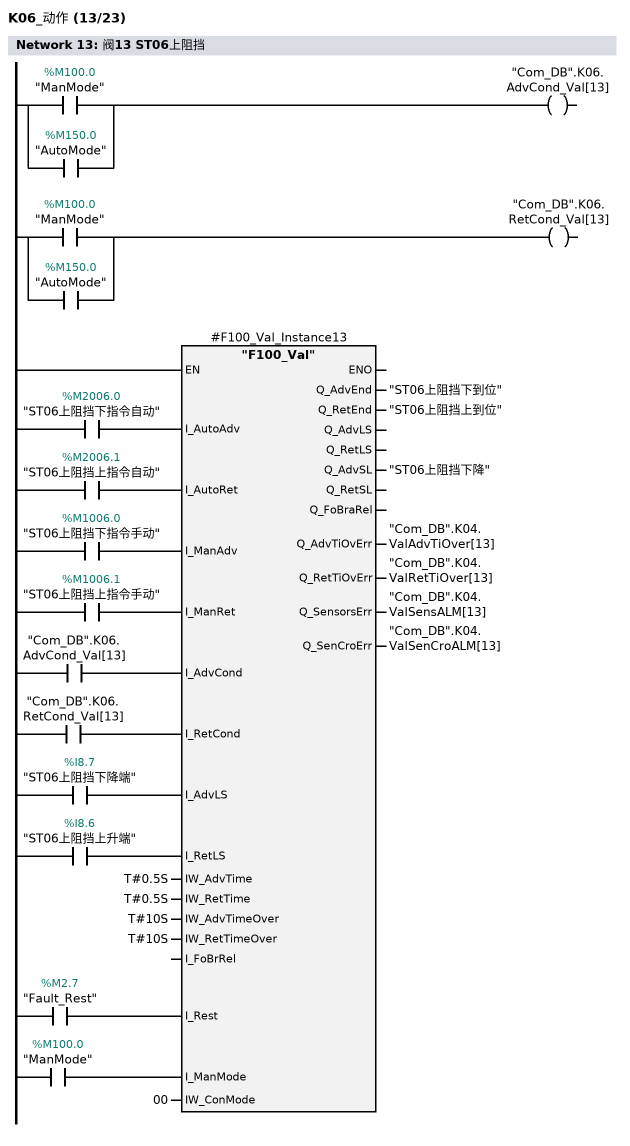
   RUNG wire#powerrail
      Contact( "ManMode" )
      wire#w1
      Coil( "Com_DB".K06.AdvCond_Val[13] )
   END_RUNG
   RUNG wire#powerrail
      Contact( "AutoMode" )
   END_RUNG wire#w1
   RUNG wire#powerrail
      Contact( "ManMode" )
      wire#w2
      Coil( "Com_DB".K06.RetCond_Val[13] )
   END_RUNG
   RUNG wire#powerrail
      Contact( "AutoMode" )
   END_RUNG wire#w2
   RUNG wire#powerrail
      #F100_Val_Instance13(I_AutoAdv := wire#w3, I_AutoRet := wire#w4, I_ManAdv := wire#w5, I_ManRet := wire#w6, I_AdvCond := wire#w7, I_RetCond := wire#w8, I_AdvLS := wire#w9, I_RetLS := wire#w10, I_Rest := wire#w11, I_ManMode := wire#w12, IW_AdvTime := T#0.5S, IW_RetTime := T#0.5S, IW_AdvTimeOver := T#10S, IW_RetTimeOver := T#10S, I_FoBrRel :=, IW_ConMode := 00, Q_AdvEnd => "ST06上阻挡下到位", Q_RetEnd => "ST06上阻挡上到位", Q_AdvLS =>, Q_RetLS =>, Q_AdvSL => "ST06上阻挡下降", Q_RetSL =>, Q_FoBraRel =>, Q_AdvTiOvErr => "Com_DB".K04.ValAdvTiOver[13], Q_RetTiOvErr => "Com_DB".K04.ValRetTiOver[13], Q_SensorsErr => "Com_DB".K04.ValSensALM[13], Q_SenCroErr => "Com_DB".K04.ValSenCroALM[13])
   END_RUNG
   RUNG wire#powerrail
      Contact( "ST06上阻挡下指令自动" )
   END_RUNG wire#w3
   RUNG wire#powerrail
      Contact( "ST06上阻挡上指令自动" )
   END_RUNG wire#w4
   RUNG wire#powerrail
      Contact( "ST06上阻挡下指令手动" )
   END_RUNG wire#w5
   RUNG wire#powerrail
      Contact( "ST06上阻挡上指令手动" )
   END_RUNG wire#w6
   RUNG wire#powerrail
      Contact( "Com_DB".K06.AdvCond_Val[13] )
   END_RUNG wire#w7
   RUNG wire#powerrail
      Contact( "Com_DB".K06.RetCond_Val[13] )
   END_RUNG wire#w8
   RUNG wire#powerrail
      Contact( "ST06上阻挡下降端" )
   END_RUNG wire#w9
   RUNG wire#powerrail
      Contact( "ST06上阻挡上升端" )
   END_RUNG wire#w10
   RUNG wire#powerrail
      Contact( "Fault_Rest" )
   END_RUNG wire#w11
   RUNG wire#powerrail
      Contact( "ManMode" )
   END_RUNG wire#w12
   // the same network as SCL:
   "Com_DB".K06.AdvCond_Val[13] := "ManMode" OR "AutoMode";
   "Com_DB".K06.RetCond_Val[13] := "ManMode" OR "AutoMode";
   #F100_Val_Instance13(I_AutoAdv := "ST06上阻挡下指令自动",   // "F100_Val"
                        I_AutoRet := "ST06上阻挡上指令自动",
                        I_ManAdv := "ST06上阻挡下指令手动",
                        I_ManRet := "ST06上阻挡上指令手动",
                        I_AdvCond := "Com_DB".K06.AdvCond_Val[13],
                        I_RetCond := "Com_DB".K06.RetCond_Val[13],
                        I_AdvLS := "ST06上阻挡下降端",
                        I_RetLS := "ST06上阻挡上升端",
                        IW_AdvTime := T#0.5S,
                        IW_RetTime := T#0.5S,
                        IW_AdvTimeOver := T#10S,
                        IW_RetTimeOver := T#10S,
                        I_Rest := "Fault_Rest",
                        I_ManMode := "ManMode",
                        IW_ConMode := 00,
                        Q_AdvEnd => "ST06上阻挡下到位",
                        Q_RetEnd => "ST06上阻挡上到位",
                        Q_AdvSL => "ST06上阻挡下降",
                        Q_AdvTiOvErr => "Com_DB".K04.ValAdvTiOver[13],
                        Q_RetTiOvErr => "Com_DB".K04.ValRetTiOver[13],
                        Q_SensorsErr => "Com_DB".K04.ValSensALM[13],
                        Q_SenCroErr => "Com_DB".K04.ValSenCroALM[13]);
END_REGION

REGION Network 14: 阀14 ST07上阻挡
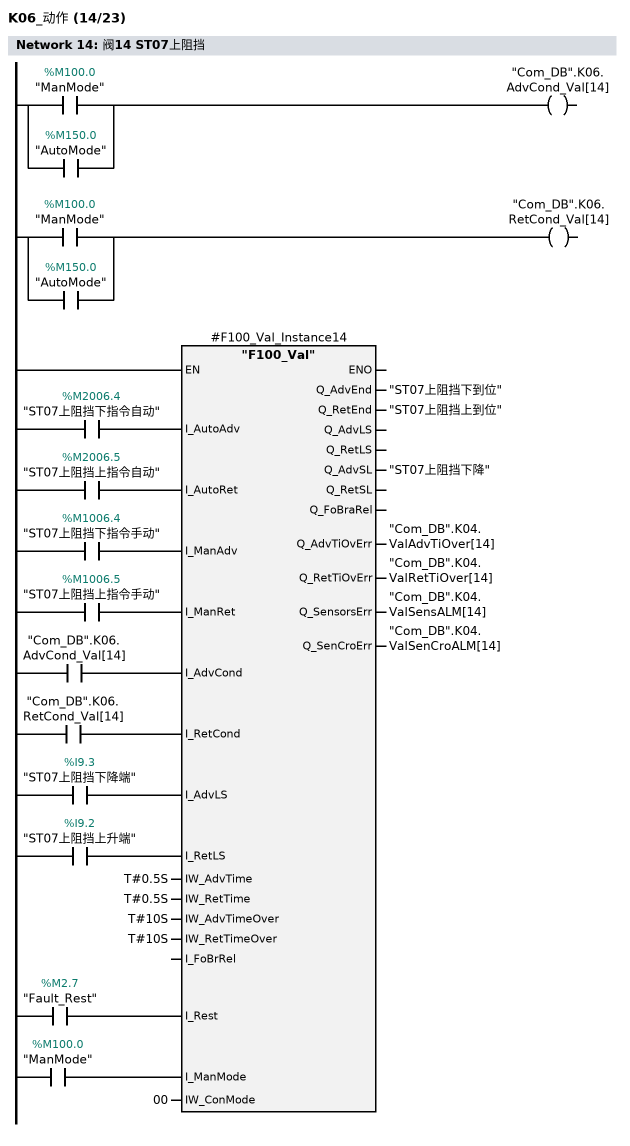
   RUNG wire#powerrail
      Contact( "ManMode" )
      wire#w1
      Coil( "Com_DB".K06.AdvCond_Val[14] )
   END_RUNG
   RUNG wire#powerrail
      Contact( "AutoMode" )
   END_RUNG wire#w1
   RUNG wire#powerrail
      Contact( "ManMode" )
      wire#w2
      Coil( "Com_DB".K06.RetCond_Val[14] )
   END_RUNG
   RUNG wire#powerrail
      Contact( "AutoMode" )
   END_RUNG wire#w2
   RUNG wire#powerrail
      #F100_Val_Instance14(I_AutoAdv := wire#w3, I_AutoRet := wire#w4, I_ManAdv := wire#w5, I_ManRet := wire#w6, I_AdvCond := wire#w7, I_RetCond := wire#w8, I_AdvLS := wire#w9, I_RetLS := wire#w10, I_Rest := wire#w11, I_ManMode := wire#w12, IW_AdvTime := T#0.5S, IW_RetTime := T#0.5S, IW_AdvTimeOver := T#10S, IW_RetTimeOver := T#10S, I_FoBrRel :=, IW_ConMode := 00, Q_AdvEnd => "ST07上阻挡下到位", Q_RetEnd => "ST07上阻挡上到位", Q_AdvLS =>, Q_RetLS =>, Q_AdvSL => "ST07上阻挡下降", Q_RetSL =>, Q_FoBraRel =>, Q_AdvTiOvErr => "Com_DB".K04.ValAdvTiOver[14], Q_RetTiOvErr => "Com_DB".K04.ValRetTiOver[14], Q_SensorsErr => "Com_DB".K04.ValSensALM[14], Q_SenCroErr => "Com_DB".K04.ValSenCroALM[14])
   END_RUNG
   RUNG wire#powerrail
      Contact( "ST07上阻挡下指令自动" )
   END_RUNG wire#w3
   RUNG wire#powerrail
      Contact( "ST07上阻挡上指令自动" )
   END_RUNG wire#w4
   RUNG wire#powerrail
      Contact( "ST07上阻挡下指令手动" )
   END_RUNG wire#w5
   RUNG wire#powerrail
      Contact( "ST07上阻挡上指令手动" )
   END_RUNG wire#w6
   RUNG wire#powerrail
      Contact( "Com_DB".K06.AdvCond_Val[14] )
   END_RUNG wire#w7
   RUNG wire#powerrail
      Contact( "Com_DB".K06.RetCond_Val[14] )
   END_RUNG wire#w8
   RUNG wire#powerrail
      Contact( "ST07上阻挡下降端" )
   END_RUNG wire#w9
   RUNG wire#powerrail
      Contact( "ST07上阻挡上升端" )
   END_RUNG wire#w10
   RUNG wire#powerrail
      Contact( "Fault_Rest" )
   END_RUNG wire#w11
   RUNG wire#powerrail
      Contact( "ManMode" )
   END_RUNG wire#w12
   // the same network as SCL:
   "Com_DB".K06.AdvCond_Val[14] := "ManMode" OR "AutoMode";
   "Com_DB".K06.RetCond_Val[14] := "ManMode" OR "AutoMode";
   #F100_Val_Instance14(I_AutoAdv := "ST07上阻挡下指令自动",   // "F100_Val"
                        I_AutoRet := "ST07上阻挡上指令自动",
                        I_ManAdv := "ST07上阻挡下指令手动",
                        I_ManRet := "ST07上阻挡上指令手动",
                        I_AdvCond := "Com_DB".K06.AdvCond_Val[14],
                        I_RetCond := "Com_DB".K06.RetCond_Val[14],
                        I_AdvLS := "ST07上阻挡下降端",
                        I_RetLS := "ST07上阻挡上升端",
                        IW_AdvTime := T#0.5S,
                        IW_RetTime := T#0.5S,
                        IW_AdvTimeOver := T#10S,
                        IW_RetTimeOver := T#10S,
                        I_Rest := "Fault_Rest",
                        I_ManMode := "ManMode",
                        IW_ConMode := 00,
                        Q_AdvEnd => "ST07上阻挡下到位",
                        Q_RetEnd => "ST07上阻挡上到位",
                        Q_AdvSL => "ST07上阻挡下降",
                        Q_AdvTiOvErr => "Com_DB".K04.ValAdvTiOver[14],
                        Q_RetTiOvErr => "Com_DB".K04.ValRetTiOver[14],
                        Q_SensorsErr => "Com_DB".K04.ValSensALM[14],
                        Q_SenCroErr => "Com_DB".K04.ValSenCroALM[14]);
END_REGION

REGION Network 15: 阀15 ST08上阻挡
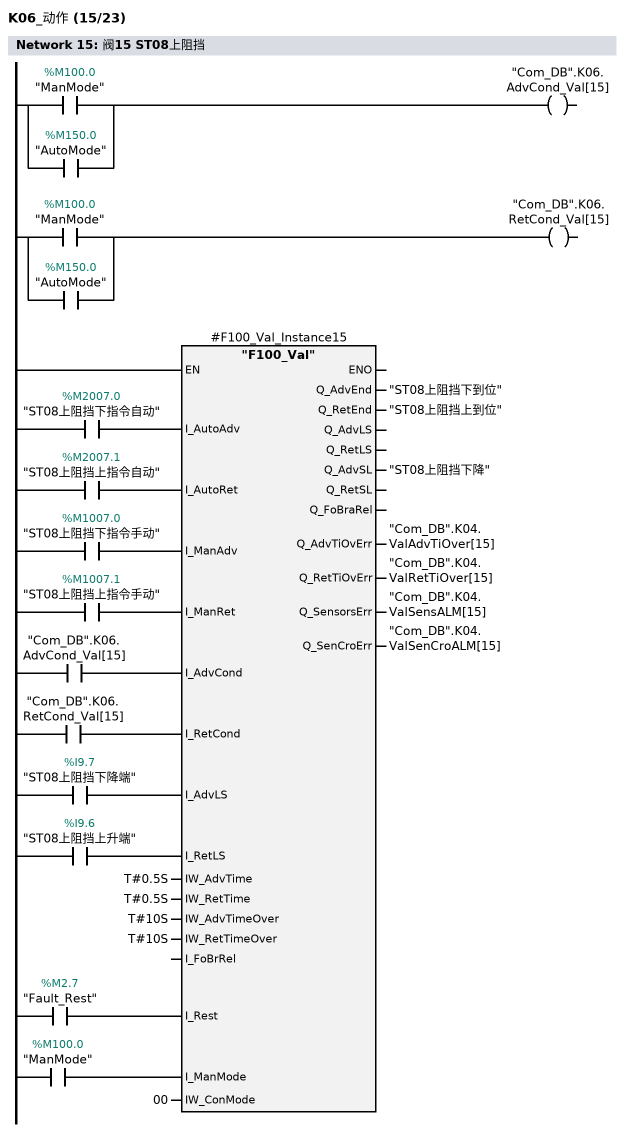
   RUNG wire#powerrail
      Contact( "ManMode" )
      wire#w1
      Coil( "Com_DB".K06.AdvCond_Val[15] )
   END_RUNG
   RUNG wire#powerrail
      Contact( "AutoMode" )
   END_RUNG wire#w1
   RUNG wire#powerrail
      Contact( "ManMode" )
      wire#w2
      Coil( "Com_DB".K06.RetCond_Val[15] )
   END_RUNG
   RUNG wire#powerrail
      Contact( "AutoMode" )
   END_RUNG wire#w2
   RUNG wire#powerrail
      #F100_Val_Instance15(I_AutoAdv := wire#w3, I_AutoRet := wire#w4, I_ManAdv := wire#w5, I_ManRet := wire#w6, I_AdvCond := wire#w7, I_RetCond := wire#w8, I_AdvLS := wire#w9, I_RetLS := wire#w10, I_Rest := wire#w11, I_ManMode := wire#w12, IW_AdvTime := T#0.5S, IW_RetTime := T#0.5S, IW_AdvTimeOver := T#10S, IW_RetTimeOver := T#10S, I_FoBrRel :=, IW_ConMode := 00, Q_AdvEnd => "ST08上阻挡下到位", Q_RetEnd => "ST08上阻挡上到位", Q_AdvLS =>, Q_RetLS =>, Q_AdvSL => "ST08上阻挡下降", Q_RetSL =>, Q_FoBraRel =>, Q_AdvTiOvErr => "Com_DB".K04.ValAdvTiOver[15], Q_RetTiOvErr => "Com_DB".K04.ValRetTiOver[15], Q_SensorsErr => "Com_DB".K04.ValSensALM[15], Q_SenCroErr => "Com_DB".K04.ValSenCroALM[15])
   END_RUNG
   RUNG wire#powerrail
      Contact( "ST08上阻挡下指令自动" )
   END_RUNG wire#w3
   RUNG wire#powerrail
      Contact( "ST08上阻挡上指令自动" )
   END_RUNG wire#w4
   RUNG wire#powerrail
      Contact( "ST08上阻挡下指令手动" )
   END_RUNG wire#w5
   RUNG wire#powerrail
      Contact( "ST08上阻挡上指令手动" )
   END_RUNG wire#w6
   RUNG wire#powerrail
      Contact( "Com_DB".K06.AdvCond_Val[15] )
   END_RUNG wire#w7
   RUNG wire#powerrail
      Contact( "Com_DB".K06.RetCond_Val[15] )
   END_RUNG wire#w8
   RUNG wire#powerrail
      Contact( "ST08上阻挡下降端" )
   END_RUNG wire#w9
   RUNG wire#powerrail
      Contact( "ST08上阻挡上升端" )
   END_RUNG wire#w10
   RUNG wire#powerrail
      Contact( "Fault_Rest" )
   END_RUNG wire#w11
   RUNG wire#powerrail
      Contact( "ManMode" )
   END_RUNG wire#w12
   // the same network as SCL:
   "Com_DB".K06.AdvCond_Val[15] := "ManMode" OR "AutoMode";
   "Com_DB".K06.RetCond_Val[15] := "ManMode" OR "AutoMode";
   #F100_Val_Instance15(I_AutoAdv := "ST08上阻挡下指令自动",   // "F100_Val"
                        I_AutoRet := "ST08上阻挡上指令自动",
                        I_ManAdv := "ST08上阻挡下指令手动",
                        I_ManRet := "ST08上阻挡上指令手动",
                        I_AdvCond := "Com_DB".K06.AdvCond_Val[15],
                        I_RetCond := "Com_DB".K06.RetCond_Val[15],
                        I_AdvLS := "ST08上阻挡下降端",
                        I_RetLS := "ST08上阻挡上升端",
                        IW_AdvTime := T#0.5S,
                        IW_RetTime := T#0.5S,
                        IW_AdvTimeOver := T#10S,
                        IW_RetTimeOver := T#10S,
                        I_Rest := "Fault_Rest",
                        I_ManMode := "ManMode",
                        IW_ConMode := 00,
                        Q_AdvEnd => "ST08上阻挡下到位",
                        Q_RetEnd => "ST08上阻挡上到位",
                        Q_AdvSL => "ST08上阻挡下降",
                        Q_AdvTiOvErr => "Com_DB".K04.ValAdvTiOver[15],
                        Q_RetTiOvErr => "Com_DB".K04.ValRetTiOver[15],
                        Q_SensorsErr => "Com_DB".K04.ValSensALM[15],
                        Q_SenCroErr => "Com_DB".K04.ValSenCroALM[15]);
END_REGION

REGION Network 16: 阀16 ST09上阻挡
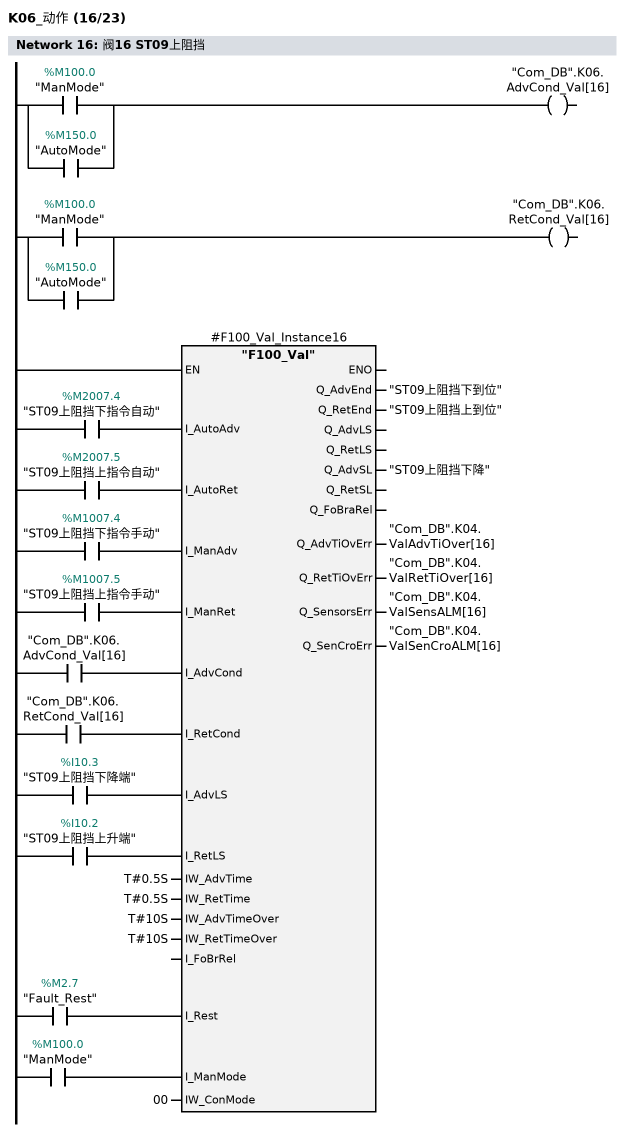
   RUNG wire#powerrail
      Contact( "ManMode" )
      wire#w1
      Coil( "Com_DB".K06.AdvCond_Val[16] )
   END_RUNG
   RUNG wire#powerrail
      Contact( "AutoMode" )
   END_RUNG wire#w1
   RUNG wire#powerrail
      Contact( "ManMode" )
      wire#w2
      Coil( "Com_DB".K06.RetCond_Val[16] )
   END_RUNG
   RUNG wire#powerrail
      Contact( "AutoMode" )
   END_RUNG wire#w2
   RUNG wire#powerrail
      #F100_Val_Instance16(I_AutoAdv := wire#w3, I_AutoRet := wire#w4, I_ManAdv := wire#w5, I_ManRet := wire#w6, I_AdvCond := wire#w7, I_RetCond := wire#w8, I_AdvLS := wire#w9, I_RetLS := wire#w10, I_Rest := wire#w11, I_ManMode := wire#w12, IW_AdvTime := T#0.5S, IW_RetTime := T#0.5S, IW_AdvTimeOver := T#10S, IW_RetTimeOver := T#10S, I_FoBrRel :=, IW_ConMode := 00, Q_AdvEnd => "ST09上阻挡下到位", Q_RetEnd => "ST09上阻挡上到位", Q_AdvLS =>, Q_RetLS =>, Q_AdvSL => "ST09上阻挡下降", Q_RetSL =>, Q_FoBraRel =>, Q_AdvTiOvErr => "Com_DB".K04.ValAdvTiOver[16], Q_RetTiOvErr => "Com_DB".K04.ValRetTiOver[16], Q_SensorsErr => "Com_DB".K04.ValSensALM[16], Q_SenCroErr => "Com_DB".K04.ValSenCroALM[16])
   END_RUNG
   RUNG wire#powerrail
      Contact( "ST09上阻挡下指令自动" )
   END_RUNG wire#w3
   RUNG wire#powerrail
      Contact( "ST09上阻挡上指令自动" )
   END_RUNG wire#w4
   RUNG wire#powerrail
      Contact( "ST09上阻挡下指令手动" )
   END_RUNG wire#w5
   RUNG wire#powerrail
      Contact( "ST09上阻挡上指令手动" )
   END_RUNG wire#w6
   RUNG wire#powerrail
      Contact( "Com_DB".K06.AdvCond_Val[16] )
   END_RUNG wire#w7
   RUNG wire#powerrail
      Contact( "Com_DB".K06.RetCond_Val[16] )
   END_RUNG wire#w8
   RUNG wire#powerrail
      Contact( "ST09上阻挡下降端" )
   END_RUNG wire#w9
   RUNG wire#powerrail
      Contact( "ST09上阻挡上升端" )
   END_RUNG wire#w10
   RUNG wire#powerrail
      Contact( "Fault_Rest" )
   END_RUNG wire#w11
   RUNG wire#powerrail
      Contact( "ManMode" )
   END_RUNG wire#w12
   // the same network as SCL:
   "Com_DB".K06.AdvCond_Val[16] := "ManMode" OR "AutoMode";
   "Com_DB".K06.RetCond_Val[16] := "ManMode" OR "AutoMode";
   #F100_Val_Instance16(I_AutoAdv := "ST09上阻挡下指令自动",   // "F100_Val"
                        I_AutoRet := "ST09上阻挡上指令自动",
                        I_ManAdv := "ST09上阻挡下指令手动",
                        I_ManRet := "ST09上阻挡上指令手动",
                        I_AdvCond := "Com_DB".K06.AdvCond_Val[16],
                        I_RetCond := "Com_DB".K06.RetCond_Val[16],
                        I_AdvLS := "ST09上阻挡下降端",
                        I_RetLS := "ST09上阻挡上升端",
                        IW_AdvTime := T#0.5S,
                        IW_RetTime := T#0.5S,
                        IW_AdvTimeOver := T#10S,
                        IW_RetTimeOver := T#10S,
                        I_Rest := "Fault_Rest",
                        I_ManMode := "ManMode",
                        IW_ConMode := 00,
                        Q_AdvEnd => "ST09上阻挡下到位",
                        Q_RetEnd => "ST09上阻挡上到位",
                        Q_AdvSL => "ST09上阻挡下降",
                        Q_AdvTiOvErr => "Com_DB".K04.ValAdvTiOver[16],
                        Q_RetTiOvErr => "Com_DB".K04.ValRetTiOver[16],
                        Q_SensorsErr => "Com_DB".K04.ValSensALM[16],
                        Q_SenCroErr => "Com_DB".K04.ValSenCroALM[16]);
END_REGION

REGION Network 17: 阀17 ST10上阻挡
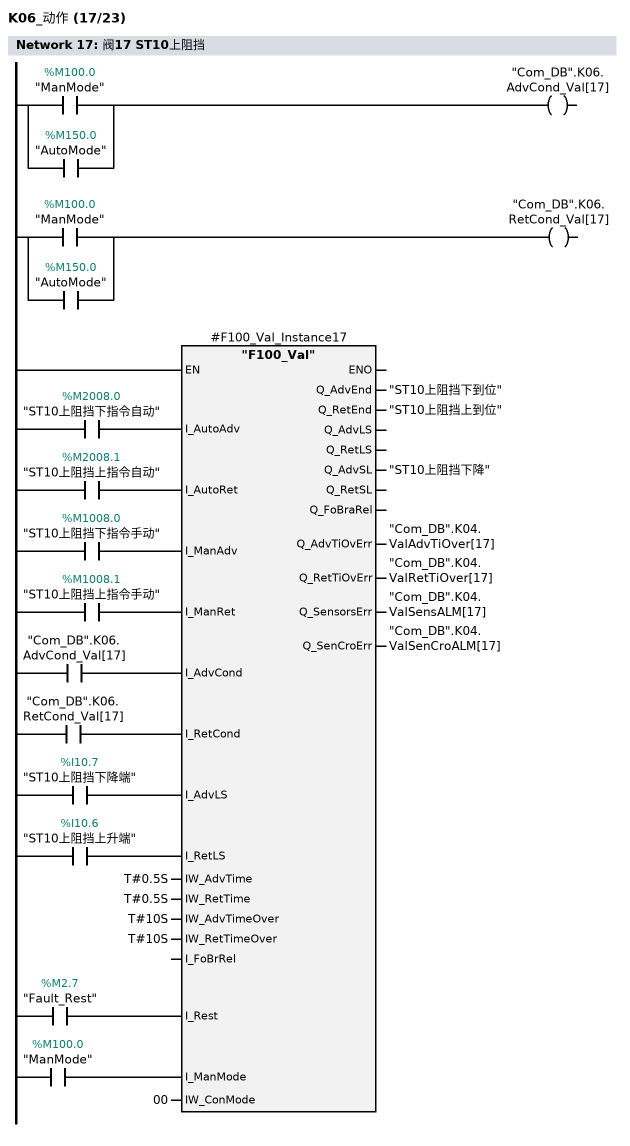
   RUNG wire#powerrail
      Contact( "ManMode" )
      wire#w1
      Coil( "Com_DB".K06.AdvCond_Val[17] )
   END_RUNG
   RUNG wire#powerrail
      Contact( "AutoMode" )
   END_RUNG wire#w1
   RUNG wire#powerrail
      Contact( "ManMode" )
      wire#w2
      Coil( "Com_DB".K06.RetCond_Val[17] )
   END_RUNG
   RUNG wire#powerrail
      Contact( "AutoMode" )
   END_RUNG wire#w2
   RUNG wire#powerrail
      #F100_Val_Instance17(I_AutoAdv := wire#w3, I_AutoRet := wire#w4, I_ManAdv := wire#w5, I_ManRet := wire#w6, I_AdvCond := wire#w7, I_RetCond := wire#w8, I_AdvLS := wire#w9, I_RetLS := wire#w10, I_Rest := wire#w11, I_ManMode := wire#w12, IW_AdvTime := T#0.5S, IW_RetTime := T#0.5S, IW_AdvTimeOver := T#10S, IW_RetTimeOver := T#10S, I_FoBrRel :=, IW_ConMode := 00, Q_AdvEnd => "ST10上阻挡下到位", Q_RetEnd => "ST10上阻挡上到位", Q_AdvLS =>, Q_RetLS =>, Q_AdvSL => "ST10上阻挡下降", Q_RetSL =>, Q_FoBraRel =>, Q_AdvTiOvErr => "Com_DB".K04.ValAdvTiOver[17], Q_RetTiOvErr => "Com_DB".K04.ValRetTiOver[17], Q_SensorsErr => "Com_DB".K04.ValSensALM[17], Q_SenCroErr => "Com_DB".K04.ValSenCroALM[17])
   END_RUNG
   RUNG wire#powerrail
      Contact( "ST10上阻挡下指令自动" )
   END_RUNG wire#w3
   RUNG wire#powerrail
      Contact( "ST10上阻挡上指令自动" )
   END_RUNG wire#w4
   RUNG wire#powerrail
      Contact( "ST10上阻挡下指令手动" )
   END_RUNG wire#w5
   RUNG wire#powerrail
      Contact( "ST10上阻挡上指令手动" )
   END_RUNG wire#w6
   RUNG wire#powerrail
      Contact( "Com_DB".K06.AdvCond_Val[17] )
   END_RUNG wire#w7
   RUNG wire#powerrail
      Contact( "Com_DB".K06.RetCond_Val[17] )
   END_RUNG wire#w8
   RUNG wire#powerrail
      Contact( "ST10上阻挡下降端" )
   END_RUNG wire#w9
   RUNG wire#powerrail
      Contact( "ST10上阻挡上升端" )
   END_RUNG wire#w10
   RUNG wire#powerrail
      Contact( "Fault_Rest" )
   END_RUNG wire#w11
   RUNG wire#powerrail
      Contact( "ManMode" )
   END_RUNG wire#w12
   // the same network as SCL:
   "Com_DB".K06.AdvCond_Val[17] := "ManMode" OR "AutoMode";
   "Com_DB".K06.RetCond_Val[17] := "ManMode" OR "AutoMode";
   #F100_Val_Instance17(I_AutoAdv := "ST10上阻挡下指令自动",   // "F100_Val"
                        I_AutoRet := "ST10上阻挡上指令自动",
                        I_ManAdv := "ST10上阻挡下指令手动",
                        I_ManRet := "ST10上阻挡上指令手动",
                        I_AdvCond := "Com_DB".K06.AdvCond_Val[17],
                        I_RetCond := "Com_DB".K06.RetCond_Val[17],
                        I_AdvLS := "ST10上阻挡下降端",
                        I_RetLS := "ST10上阻挡上升端",
                        IW_AdvTime := T#0.5S,
                        IW_RetTime := T#0.5S,
                        IW_AdvTimeOver := T#10S,
                        IW_RetTimeOver := T#10S,
                        I_Rest := "Fault_Rest",
                        I_ManMode := "ManMode",
                        IW_ConMode := 00,
                        Q_AdvEnd => "ST10上阻挡下到位",
                        Q_RetEnd => "ST10上阻挡上到位",
                        Q_AdvSL => "ST10上阻挡下降",
                        Q_AdvTiOvErr => "Com_DB".K04.ValAdvTiOver[17],
                        Q_RetTiOvErr => "Com_DB".K04.ValRetTiOver[17],
                        Q_SensorsErr => "Com_DB".K04.ValSensALM[17],
                        Q_SenCroErr => "Com_DB".K04.ValSenCroALM[17]);
END_REGION

REGION Network 18: 阀18 ST11上阻挡
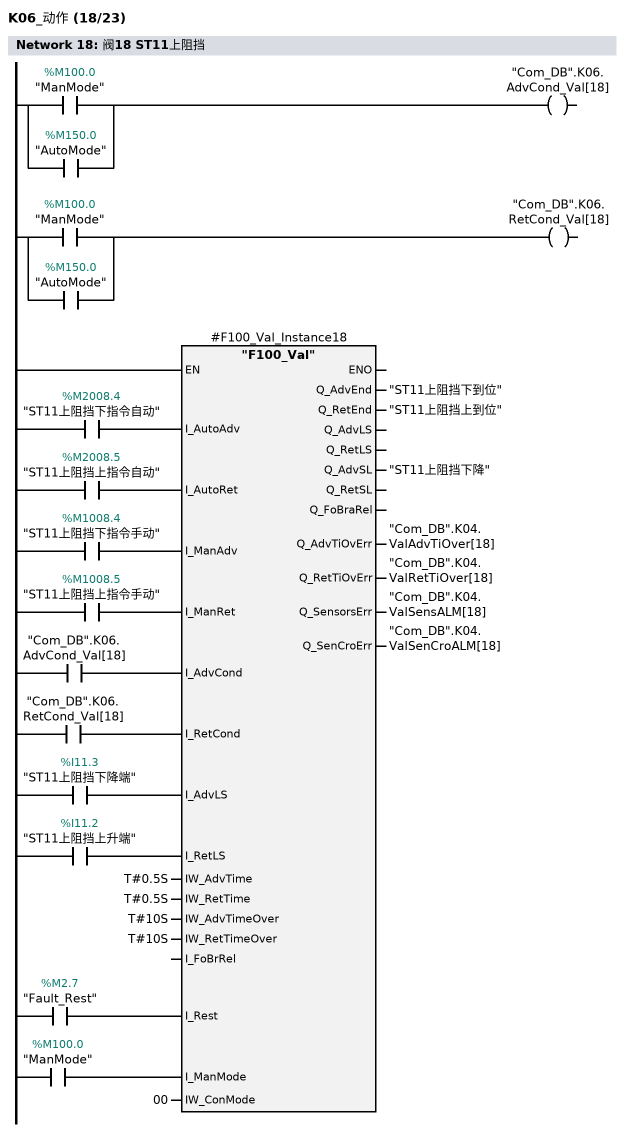
   RUNG wire#powerrail
      Contact( "ManMode" )
      wire#w1
      Coil( "Com_DB".K06.AdvCond_Val[18] )
   END_RUNG
   RUNG wire#powerrail
      Contact( "AutoMode" )
   END_RUNG wire#w1
   RUNG wire#powerrail
      Contact( "ManMode" )
      wire#w2
      Coil( "Com_DB".K06.RetCond_Val[18] )
   END_RUNG
   RUNG wire#powerrail
      Contact( "AutoMode" )
   END_RUNG wire#w2
   RUNG wire#powerrail
      #F100_Val_Instance18(I_AutoAdv := wire#w3, I_AutoRet := wire#w4, I_ManAdv := wire#w5, I_ManRet := wire#w6, I_AdvCond := wire#w7, I_RetCond := wire#w8, I_AdvLS := wire#w9, I_RetLS := wire#w10, I_Rest := wire#w11, I_ManMode := wire#w12, IW_AdvTime := T#0.5S, IW_RetTime := T#0.5S, IW_AdvTimeOver := T#10S, IW_RetTimeOver := T#10S, I_FoBrRel :=, IW_ConMode := 00, Q_AdvEnd => "ST11上阻挡下到位", Q_RetEnd => "ST11上阻挡上到位", Q_AdvLS =>, Q_RetLS =>, Q_AdvSL => "ST11上阻挡下降", Q_RetSL =>, Q_FoBraRel =>, Q_AdvTiOvErr => "Com_DB".K04.ValAdvTiOver[18], Q_RetTiOvErr => "Com_DB".K04.ValRetTiOver[18], Q_SensorsErr => "Com_DB".K04.ValSensALM[18], Q_SenCroErr => "Com_DB".K04.ValSenCroALM[18])
   END_RUNG
   RUNG wire#powerrail
      Contact( "ST11上阻挡下指令自动" )
   END_RUNG wire#w3
   RUNG wire#powerrail
      Contact( "ST11上阻挡上指令自动" )
   END_RUNG wire#w4
   RUNG wire#powerrail
      Contact( "ST11上阻挡下指令手动" )
   END_RUNG wire#w5
   RUNG wire#powerrail
      Contact( "ST11上阻挡上指令手动" )
   END_RUNG wire#w6
   RUNG wire#powerrail
      Contact( "Com_DB".K06.AdvCond_Val[18] )
   END_RUNG wire#w7
   RUNG wire#powerrail
      Contact( "Com_DB".K06.RetCond_Val[18] )
   END_RUNG wire#w8
   RUNG wire#powerrail
      Contact( "ST11上阻挡下降端" )
   END_RUNG wire#w9
   RUNG wire#powerrail
      Contact( "ST11上阻挡上升端" )
   END_RUNG wire#w10
   RUNG wire#powerrail
      Contact( "Fault_Rest" )
   END_RUNG wire#w11
   RUNG wire#powerrail
      Contact( "ManMode" )
   END_RUNG wire#w12
   // the same network as SCL:
   "Com_DB".K06.AdvCond_Val[18] := "ManMode" OR "AutoMode";
   "Com_DB".K06.RetCond_Val[18] := "ManMode" OR "AutoMode";
   #F100_Val_Instance18(I_AutoAdv := "ST11上阻挡下指令自动",   // "F100_Val"
                        I_AutoRet := "ST11上阻挡上指令自动",
                        I_ManAdv := "ST11上阻挡下指令手动",
                        I_ManRet := "ST11上阻挡上指令手动",
                        I_AdvCond := "Com_DB".K06.AdvCond_Val[18],
                        I_RetCond := "Com_DB".K06.RetCond_Val[18],
                        I_AdvLS := "ST11上阻挡下降端",
                        I_RetLS := "ST11上阻挡上升端",
                        IW_AdvTime := T#0.5S,
                        IW_RetTime := T#0.5S,
                        IW_AdvTimeOver := T#10S,
                        IW_RetTimeOver := T#10S,
                        I_Rest := "Fault_Rest",
                        I_ManMode := "ManMode",
                        IW_ConMode := 00,
                        Q_AdvEnd => "ST11上阻挡下到位",
                        Q_RetEnd => "ST11上阻挡上到位",
                        Q_AdvSL => "ST11上阻挡下降",
                        Q_AdvTiOvErr => "Com_DB".K04.ValAdvTiOver[18],
                        Q_RetTiOvErr => "Com_DB".K04.ValRetTiOver[18],
                        Q_SensorsErr => "Com_DB".K04.ValSensALM[18],
                        Q_SenCroErr => "Com_DB".K04.ValSenCroALM[18]);
END_REGION

REGION Network 19: 阀19 ST12上阻挡
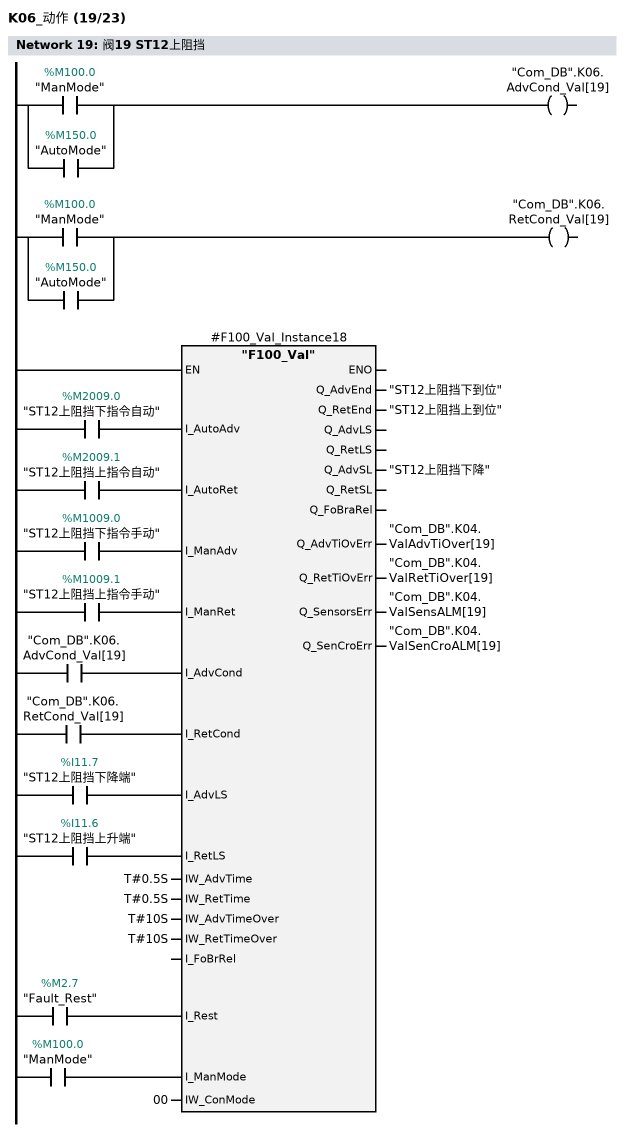
   RUNG wire#powerrail
      Contact( "ManMode" )
      wire#w1
      Coil( "Com_DB".K06.AdvCond_Val[19] )
   END_RUNG
   RUNG wire#powerrail
      Contact( "AutoMode" )
   END_RUNG wire#w1
   RUNG wire#powerrail
      Contact( "ManMode" )
      wire#w2
      Coil( "Com_DB".K06.RetCond_Val[19] )
   END_RUNG
   RUNG wire#powerrail
      Contact( "AutoMode" )
   END_RUNG wire#w2
   RUNG wire#powerrail
      #F100_Val_Instance18(I_AutoAdv := wire#w3, I_AutoRet := wire#w4, I_ManAdv := wire#w5, I_ManRet := wire#w6, I_AdvCond := wire#w7, I_RetCond := wire#w8, I_AdvLS := wire#w9, I_RetLS := wire#w10, I_Rest := wire#w11, I_ManMode := wire#w12, IW_AdvTime := T#0.5S, IW_RetTime := T#0.5S, IW_AdvTimeOver := T#10S, IW_RetTimeOver := T#10S, I_FoBrRel :=, IW_ConMode := 00, Q_AdvEnd => "ST12上阻挡下到位", Q_RetEnd => "ST12上阻挡上到位", Q_AdvLS =>, Q_RetLS =>, Q_AdvSL => "ST12上阻挡下降", Q_RetSL =>, Q_FoBraRel =>, Q_AdvTiOvErr => "Com_DB".K04.ValAdvTiOver[19], Q_RetTiOvErr => "Com_DB".K04.ValRetTiOver[19], Q_SensorsErr => "Com_DB".K04.ValSensALM[19], Q_SenCroErr => "Com_DB".K04.ValSenCroALM[19])
   END_RUNG
   RUNG wire#powerrail
      Contact( "ST12上阻挡下指令自动" )
   END_RUNG wire#w3
   RUNG wire#powerrail
      Contact( "ST12上阻挡上指令自动" )
   END_RUNG wire#w4
   RUNG wire#powerrail
      Contact( "ST12上阻挡下指令手动" )
   END_RUNG wire#w5
   RUNG wire#powerrail
      Contact( "ST12上阻挡上指令手动" )
   END_RUNG wire#w6
   RUNG wire#powerrail
      Contact( "Com_DB".K06.AdvCond_Val[19] )
   END_RUNG wire#w7
   RUNG wire#powerrail
      Contact( "Com_DB".K06.RetCond_Val[19] )
   END_RUNG wire#w8
   RUNG wire#powerrail
      Contact( "ST12上阻挡下降端" )
   END_RUNG wire#w9
   RUNG wire#powerrail
      Contact( "ST12上阻挡上升端" )
   END_RUNG wire#w10
   RUNG wire#powerrail
      Contact( "Fault_Rest" )
   END_RUNG wire#w11
   RUNG wire#powerrail
      Contact( "ManMode" )
   END_RUNG wire#w12
   // the same network as SCL:
   "Com_DB".K06.AdvCond_Val[19] := "ManMode" OR "AutoMode";
   "Com_DB".K06.RetCond_Val[19] := "ManMode" OR "AutoMode";
   #F100_Val_Instance18(I_AutoAdv := "ST12上阻挡下指令自动",   // "F100_Val"
                        I_AutoRet := "ST12上阻挡上指令自动",
                        I_ManAdv := "ST12上阻挡下指令手动",
                        I_ManRet := "ST12上阻挡上指令手动",
                        I_AdvCond := "Com_DB".K06.AdvCond_Val[19],
                        I_RetCond := "Com_DB".K06.RetCond_Val[19],
                        I_AdvLS := "ST12上阻挡下降端",
                        I_RetLS := "ST12上阻挡上升端",
                        IW_AdvTime := T#0.5S,
                        IW_RetTime := T#0.5S,
                        IW_AdvTimeOver := T#10S,
                        IW_RetTimeOver := T#10S,
                        I_Rest := "Fault_Rest",
                        I_ManMode := "ManMode",
                        IW_ConMode := 00,
                        Q_AdvEnd => "ST12上阻挡下到位",
                        Q_RetEnd => "ST12上阻挡上到位",
                        Q_AdvSL => "ST12上阻挡下降",
                        Q_AdvTiOvErr => "Com_DB".K04.ValAdvTiOver[19],
                        Q_RetTiOvErr => "Com_DB".K04.ValRetTiOver[19],
                        Q_SensorsErr => "Com_DB".K04.ValSensALM[19],
                        Q_SenCroErr => "Com_DB".K04.ValSenCroALM[19]);
END_REGION

REGION Network 20: 变频器1-入口搬送电机
   // 滚筒控制也可以使用变频器FB库，正转上层送托盘，反转下层接托盘
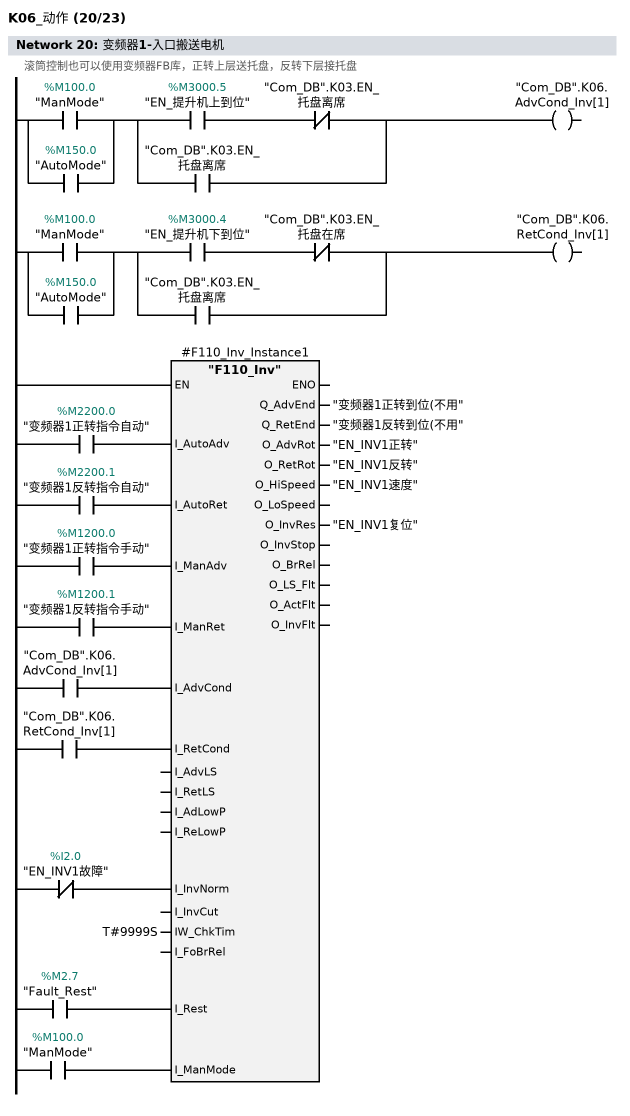
   RUNG wire#powerrail
      Contact( "ManMode" )
      wire#w1
      Contact( "EN_提升机上到位" )
      I_Contact( "Com_DB".K03.EN_托盘离席 )
      wire#w2
      Coil( "Com_DB".K06.AdvCond_Inv[1] )
   END_RUNG
   RUNG wire#powerrail
      Contact( "AutoMode" )
   END_RUNG wire#w1
   RUNG wire#w1
      Contact( "Com_DB".K03.EN_托盘离席 )
   END_RUNG wire#w2
   RUNG wire#powerrail
      Contact( "ManMode" )
      wire#w3
      Contact( "EN_提升机下到位" )
      I_Contact( "Com_DB".K03.EN_托盘在席 )
      wire#w4
      Coil( "Com_DB".K06.RetCond_Inv[1] )
   END_RUNG
   RUNG wire#powerrail
      Contact( "AutoMode" )
   END_RUNG wire#w3
   RUNG wire#w3
      Contact( "Com_DB".K03.EN_托盘离席 )
   END_RUNG wire#w4
   RUNG wire#powerrail
      #F110_Inv_Instance1(I_AutoAdv := wire#w5, I_AutoRet := wire#w6, I_ManAdv := wire#w7, I_ManRet := wire#w8, I_AdvCond := wire#w9, I_RetCond := wire#w10, I_InvNorm := wire#w11, I_Rest := wire#w12, I_ManMode := wire#w13, I_AdvLS :=, I_RetLS :=, I_AdLowP :=, I_ReLowP :=, I_InvCut :=, IW_ChkTim := T#9999S, I_FoBrRel :=, Q_AdvEnd => "变频器1正转到位(不用", Q_RetEnd => "变频器1反转到位(不用", O_AdvRot => "EN_INV1正转", O_RetRot => "EN_INV1反转", O_HiSpeed => "EN_INV1速度", O_LoSpeed =>, O_InvRes => "EN_INV1复位", O_InvStop =>, O_BrRel =>, O_LS_Flt =>, O_ActFlt =>, O_InvFlt =>)
   END_RUNG
   RUNG wire#powerrail
      Contact( "变频器1正转指令自动" )
   END_RUNG wire#w5
   RUNG wire#powerrail
      Contact( "变频器1反转指令自动" )
   END_RUNG wire#w6
   RUNG wire#powerrail
      Contact( "变频器1正转指令手动" )
   END_RUNG wire#w7
   RUNG wire#powerrail
      Contact( "变频器1反转指令手动" )
   END_RUNG wire#w8
   RUNG wire#powerrail
      Contact( "Com_DB".K06.AdvCond_Inv[1] )
   END_RUNG wire#w9
   RUNG wire#powerrail
      Contact( "Com_DB".K06.RetCond_Inv[1] )
   END_RUNG wire#w10
   RUNG wire#powerrail
      I_Contact( "EN_INV1故障" )
   END_RUNG wire#w11
   RUNG wire#powerrail
      Contact( "Fault_Rest" )
   END_RUNG wire#w12
   RUNG wire#powerrail
      Contact( "ManMode" )
   END_RUNG wire#w13
   // the same network as SCL:
   "Com_DB".K06.AdvCond_Inv[1] := ("ManMode" OR "AutoMode") AND (("EN_提升机上到位" AND NOT "Com_DB".K03.EN_托盘离席) OR "Com_DB".K03.EN_托盘离席);
   "Com_DB".K06.RetCond_Inv[1] := ("ManMode" OR "AutoMode") AND (("EN_提升机下到位" AND NOT "Com_DB".K03.EN_托盘在席) OR "Com_DB".K03.EN_托盘离席);
   #F110_Inv_Instance1(I_AutoAdv := "变频器1正转指令自动",   // "F110_Inv"
                       I_AutoRet := "变频器1反转指令自动",
                       I_ManAdv := "变频器1正转指令手动",
                       I_ManRet := "变频器1反转指令手动",
                       I_AdvCond := "Com_DB".K06.AdvCond_Inv[1],
                       I_RetCond := "Com_DB".K06.RetCond_Inv[1],
                       I_InvNorm := NOT "EN_INV1故障",
                       IW_ChkTim := T#9999S,
                       I_Rest := "Fault_Rest",
                       I_ManMode := "ManMode",
                       Q_AdvEnd => "变频器1正转到位(不用",
                       Q_RetEnd => "变频器1反转到位(不用",
                       O_AdvRot => "EN_INV1正转",
                       O_RetRot => "EN_INV1反转",
                       O_HiSpeed => "EN_INV1速度",
                       O_InvRes => "EN_INV1复位");
END_REGION

REGION Network 21: 变频器2 出口搬送电机
   // 正转上层J接托盘，反转下层送托盘
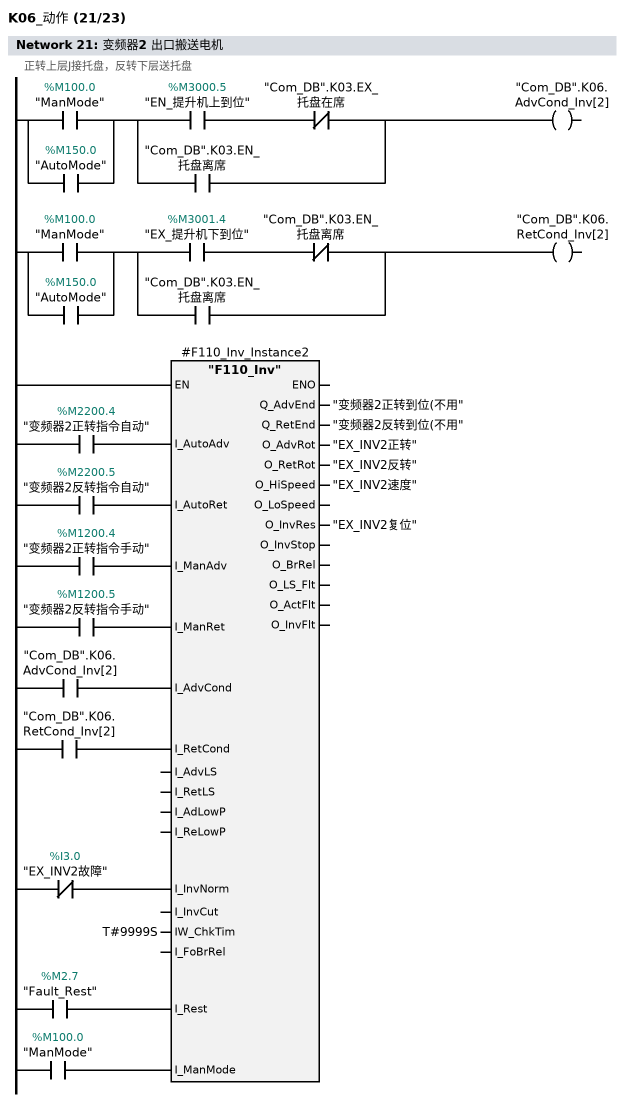
   RUNG wire#powerrail
      Contact( "ManMode" )
      wire#w1
      Contact( "EN_提升机上到位" )
      I_Contact( "Com_DB".K03.EX_托盘在席 )
      wire#w2
      Coil( "Com_DB".K06.AdvCond_Inv[2] )
   END_RUNG
   RUNG wire#powerrail
      Contact( "AutoMode" )
   END_RUNG wire#w1
   RUNG wire#w1
      Contact( "Com_DB".K03.EN_托盘离席 )
   END_RUNG wire#w2
   RUNG wire#powerrail
      Contact( "ManMode" )
      wire#w3
      Contact( "EX_提升机下到位" )
      I_Contact( "Com_DB".K03.EN_托盘离席 )
      wire#w4
      Coil( "Com_DB".K06.RetCond_Inv[2] )
   END_RUNG
   RUNG wire#powerrail
      Contact( "AutoMode" )
   END_RUNG wire#w3
   RUNG wire#w3
      Contact( "Com_DB".K03.EN_托盘离席 )
   END_RUNG wire#w4
   RUNG wire#powerrail
      #F110_Inv_Instance2(I_AutoAdv := wire#w5, I_AutoRet := wire#w6, I_ManAdv := wire#w7, I_ManRet := wire#w8, I_AdvCond := wire#w9, I_RetCond := wire#w10, I_InvNorm := wire#w11, I_Rest := wire#w12, I_ManMode := wire#w13, I_AdvLS :=, I_RetLS :=, I_AdLowP :=, I_ReLowP :=, I_InvCut :=, IW_ChkTim := T#9999S, I_FoBrRel :=, Q_AdvEnd => "变频器2正转到位(不用", Q_RetEnd => "变频器2反转到位(不用", O_AdvRot => "EX_INV2正转", O_RetRot => "EX_INV2反转", O_HiSpeed => "EX_INV2速度", O_LoSpeed =>, O_InvRes => "EX_INV2复位", O_InvStop =>, O_BrRel =>, O_LS_Flt =>, O_ActFlt =>, O_InvFlt =>)
   END_RUNG
   RUNG wire#powerrail
      Contact( "变频器2正转指令自动" )
   END_RUNG wire#w5
   RUNG wire#powerrail
      Contact( "变频器2反转指令自动" )
   END_RUNG wire#w6
   RUNG wire#powerrail
      Contact( "变频器2正转指令手动" )
   END_RUNG wire#w7
   RUNG wire#powerrail
      Contact( "变频器2反转指令手动" )
   END_RUNG wire#w8
   RUNG wire#powerrail
      Contact( "Com_DB".K06.AdvCond_Inv[2] )
   END_RUNG wire#w9
   RUNG wire#powerrail
      Contact( "Com_DB".K06.RetCond_Inv[2] )
   END_RUNG wire#w10
   RUNG wire#powerrail
      I_Contact( "EX_INV2故障" )
   END_RUNG wire#w11
   RUNG wire#powerrail
      Contact( "Fault_Rest" )
   END_RUNG wire#w12
   RUNG wire#powerrail
      Contact( "ManMode" )
   END_RUNG wire#w13
   // the same network as SCL:
   "Com_DB".K06.AdvCond_Inv[2] := ("ManMode" OR "AutoMode") AND (("EN_提升机上到位" AND NOT "Com_DB".K03.EX_托盘在席) OR "Com_DB".K03.EN_托盘离席);
   "Com_DB".K06.RetCond_Inv[2] := ("ManMode" OR "AutoMode") AND (("EX_提升机下到位" AND NOT "Com_DB".K03.EN_托盘离席) OR "Com_DB".K03.EN_托盘离席);
   #F110_Inv_Instance2(I_AutoAdv := "变频器2正转指令自动",   // "F110_Inv"
                       I_AutoRet := "变频器2反转指令自动",
                       I_ManAdv := "变频器2正转指令手动",
                       I_ManRet := "变频器2反转指令手动",
                       I_AdvCond := "Com_DB".K06.AdvCond_Inv[2],
                       I_RetCond := "Com_DB".K06.RetCond_Inv[2],
                       I_InvNorm := NOT "EX_INV2故障",
                       IW_ChkTim := T#9999S,
                       I_Rest := "Fault_Rest",
                       I_ManMode := "ManMode",
                       Q_AdvEnd => "变频器2正转到位(不用",
                       Q_RetEnd => "变频器2反转到位(不用",
                       O_AdvRot => "EX_INV2正转",
                       O_RetRot => "EX_INV2反转",
                       O_HiSpeed => "EX_INV2速度",
                       O_InvRes => "EX_INV2复位");
END_REGION

REGION Network 22: 变频器3/5 前段/后段上层搬送电机，因为上层变频器条件一致，功能一致。共用1个FB
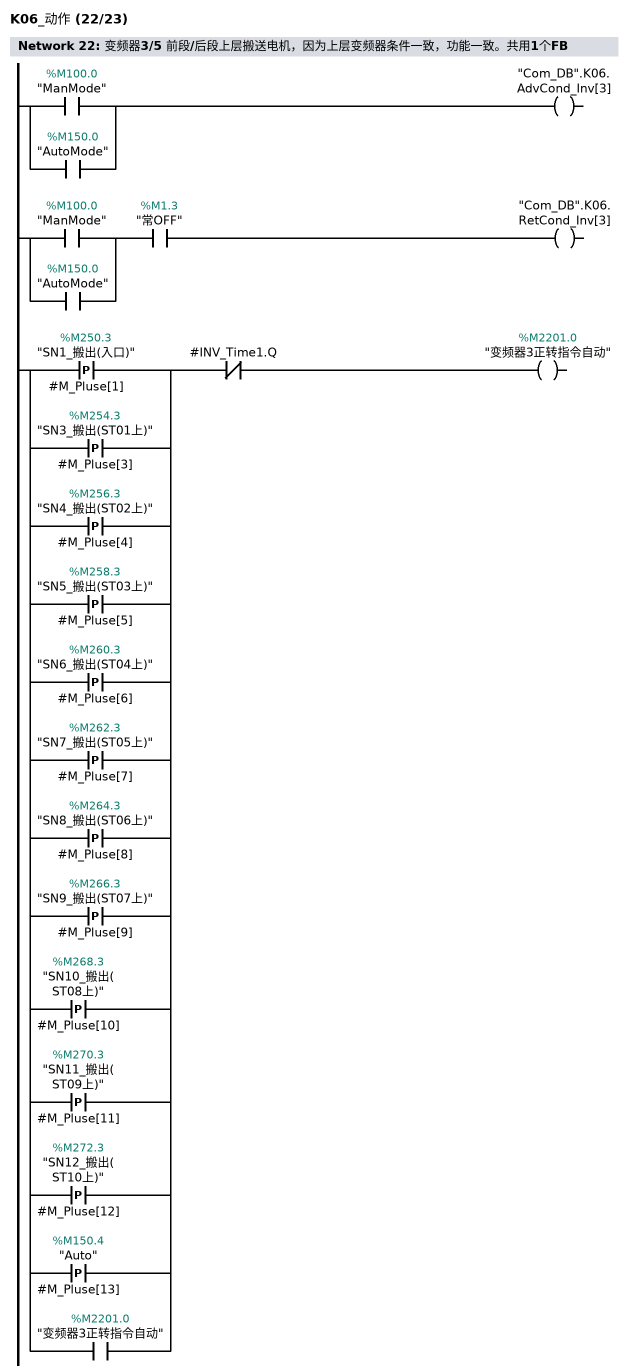
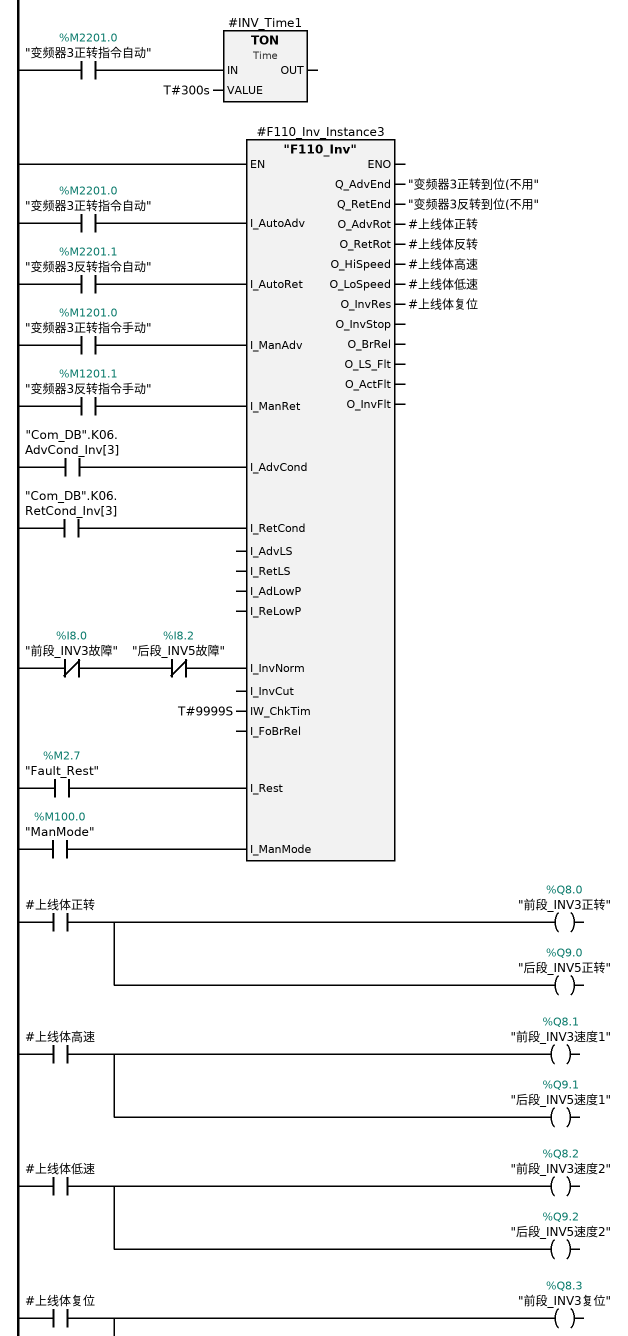
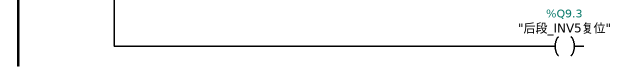
   "Com_DB".K06.AdvCond_Inv[3] := "ManMode" OR "AutoMode";
   "Com_DB".K06.RetCond_Inv[3] := ("ManMode" OR "AutoMode") AND "常OFF";
   #_w1 := "SN1_搬出(入口)" AND NOT #M_Pluse[1];   // rising edge of "SN1_搬出(入口)"
   #M_Pluse[1] := "SN1_搬出(入口)";
   #_w2 := "SN3_搬出(ST01上)" AND NOT #M_Pluse[3];   // rising edge of "SN3_搬出(ST01上)"
   #M_Pluse[3] := "SN3_搬出(ST01上)";
   #_w3 := "SN4_搬出(ST02上)" AND NOT #M_Pluse[4];   // rising edge of "SN4_搬出(ST02上)"
   #M_Pluse[4] := "SN4_搬出(ST02上)";
   #_w4 := "SN5_搬出(ST03上)" AND NOT #M_Pluse[5];   // rising edge of "SN5_搬出(ST03上)"
   #M_Pluse[5] := "SN5_搬出(ST03上)";
   #_w5 := "SN6_搬出(ST04上)" AND NOT #M_Pluse[6];   // rising edge of "SN6_搬出(ST04上)"
   #M_Pluse[6] := "SN6_搬出(ST04上)";
   #_w6 := "SN7_搬出(ST05上)" AND NOT #M_Pluse[7];   // rising edge of "SN7_搬出(ST05上)"
   #M_Pluse[7] := "SN7_搬出(ST05上)";
   #_w7 := "SN8_搬出(ST06上)" AND NOT #M_Pluse[8];   // rising edge of "SN8_搬出(ST06上)"
   #M_Pluse[8] := "SN8_搬出(ST06上)";
   #_w8 := "SN9_搬出(ST07上)" AND NOT #M_Pluse[9];   // rising edge of "SN9_搬出(ST07上)"
   #M_Pluse[9] := "SN9_搬出(ST07上)";
   #_w9 := "SN10_搬出(ST08上)" AND NOT #M_Pluse[10];   // rising edge of "SN10_搬出(ST08上)"
   #M_Pluse[10] := "SN10_搬出(ST08上)";
   #_w10 := "SN11_搬出(ST09上)" AND NOT #M_Pluse[11];   // rising edge of "SN11_搬出(ST09上)"
   #M_Pluse[11] := "SN11_搬出(ST09上)";
   #_w11 := "SN12_搬出(ST10上)" AND NOT #M_Pluse[12];   // rising edge of "SN12_搬出(ST10上)"
   #M_Pluse[12] := "SN12_搬出(ST10上)";
   #_w12 := "Auto" AND NOT #M_Pluse[13];   // rising edge of "Auto"
   #M_Pluse[13] := "Auto";
   "变频器3正转指令自动" := (#_w1 OR #_w2 OR #_w3 OR #_w4 OR #_w5 OR #_w6 OR #_w7 OR #_w8 OR #_w9 OR #_w10 OR #_w11 OR #_w12 OR "变频器3正转指令自动") AND NOT #INV_Time1.Q;
   #INV_Time1.TON(IN := "变频器3正转指令自动", PT := T#300s);   // TON coil
   #F110_Inv_Instance3(I_AutoAdv := "变频器3正转指令自动",   // "F110_Inv"
                       I_AutoRet := "变频器3反转指令自动",
                       I_ManAdv := "变频器3正转指令手动",
                       I_ManRet := "变频器3反转指令手动",
                       I_AdvCond := "Com_DB".K06.AdvCond_Inv[3],
                       I_RetCond := "Com_DB".K06.RetCond_Inv[3],
                       I_InvNorm := NOT "前段_INV3故障" AND NOT "后段_INV5故障",
                       IW_ChkTim := T#9999S,
                       I_Rest := "Fault_Rest",
                       I_ManMode := "ManMode",
                       Q_AdvEnd => "变频器3正转到位(不用",
                       Q_RetEnd => "变频器3反转到位(不用",
                       O_AdvRot => #上线体正转,
                       O_RetRot => #上线体反转,
                       O_HiSpeed => #上线体高速,
                       O_LoSpeed => #上线体低速,
                       O_InvRes => #上线体复位);
   "前段_INV3正转" := #上线体正转;
   "后段_INV5正转" := #上线体正转;
   "前段_INV3速度1" := #上线体高速;
   "后段_INV5速度1" := #上线体高速;
   "前段_INV3速度2" := #上线体低速;
   "后段_INV5速度2" := #上线体低速;
   "前段_INV3复位" := #上线体复位;
   "后段_INV5复位" := #上线体复位;
END_REGION

REGION Network 23: 变频器4/6前段/后段下层搬送电机。因为上层变频器条件一致，功能一致。共用1个FB
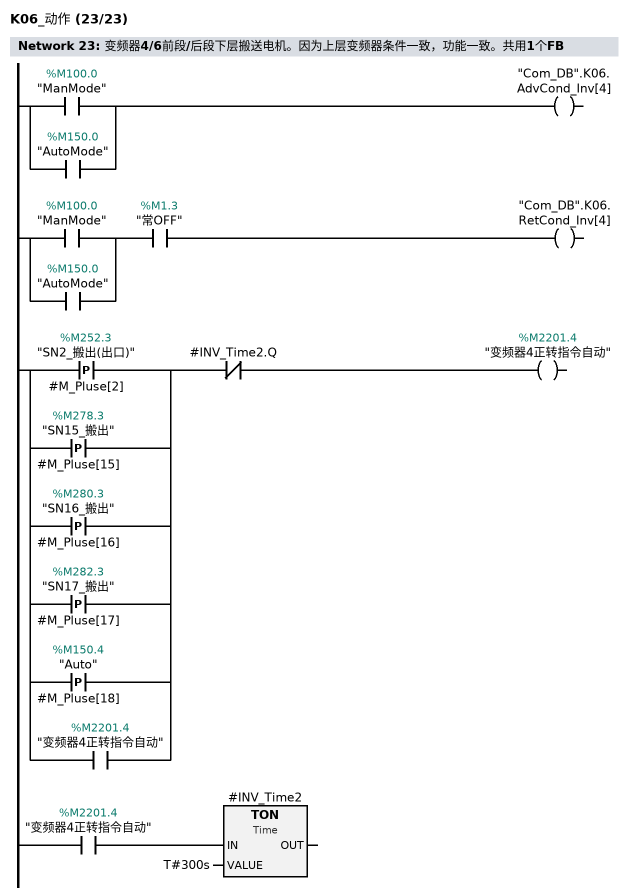
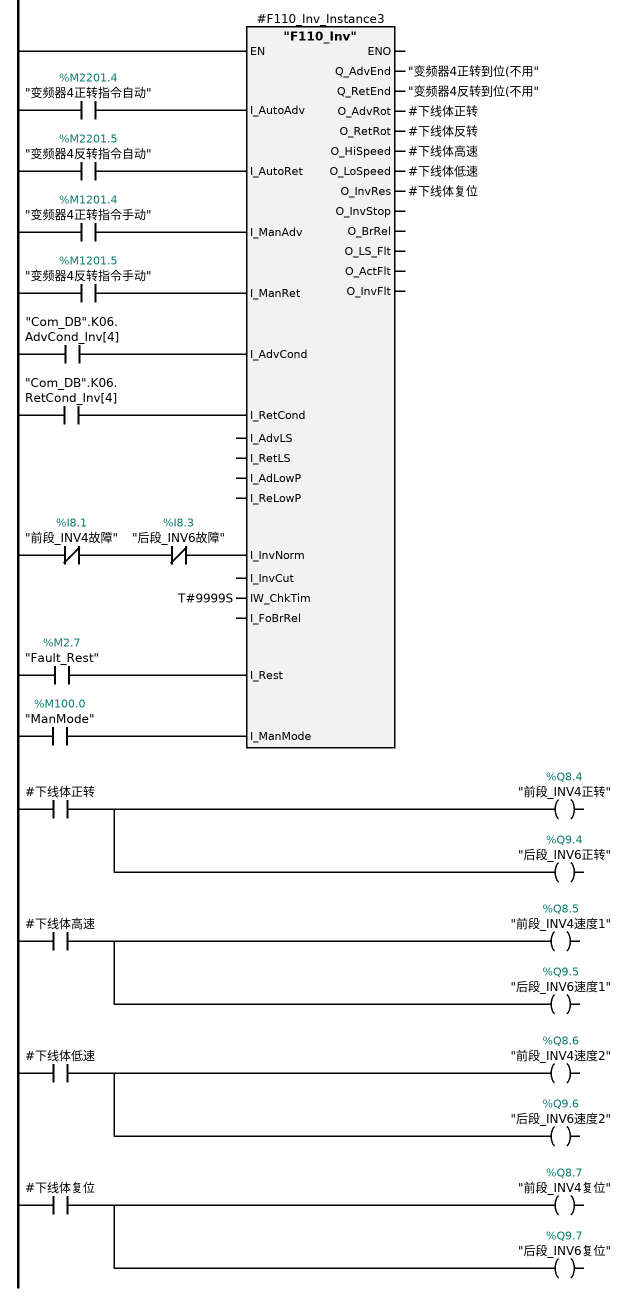
   "Com_DB".K06.AdvCond_Inv[4] := "ManMode" OR "AutoMode";
   "Com_DB".K06.RetCond_Inv[4] := ("ManMode" OR "AutoMode") AND "常OFF";
   #_w1 := "SN2_搬出(出口)" AND NOT #M_Pluse[2];   // rising edge of "SN2_搬出(出口)"
   #M_Pluse[2] := "SN2_搬出(出口)";
   #_w2 := "SN15_搬出" AND NOT #M_Pluse[15];   // rising edge of "SN15_搬出"
   #M_Pluse[15] := "SN15_搬出";
   #_w3 := "SN16_搬出" AND NOT #M_Pluse[16];   // rising edge of "SN16_搬出"
   #M_Pluse[16] := "SN16_搬出";
   #_w4 := "SN17_搬出" AND NOT #M_Pluse[17];   // rising edge of "SN17_搬出"
   #M_Pluse[17] := "SN17_搬出";
   #_w5 := "Auto" AND NOT #M_Pluse[18];   // rising edge of "Auto"
   #M_Pluse[18] := "Auto";
   "变频器4正转指令自动" := (#_w1 OR #_w2 OR #_w3 OR #_w4 OR #_w5 OR "变频器4正转指令自动") AND NOT #INV_Time2.Q;
   #INV_Time2.TON(IN := "变频器4正转指令自动", PT := T#300s);   // TON coil
   #F110_Inv_Instance3(I_AutoAdv := "变频器4正转指令自动",   // "F110_Inv"
                       I_AutoRet := "变频器4反转指令自动",
                       I_ManAdv := "变频器4正转指令手动",
                       I_ManRet := "变频器4反转指令手动",
                       I_AdvCond := "Com_DB".K06.AdvCond_Inv[4],
                       I_RetCond := "Com_DB".K06.RetCond_Inv[4],
                       I_InvNorm := NOT "前段_INV4故障" AND NOT "后段_INV6故障",
                       IW_ChkTim := T#9999S,
                       I_Rest := "Fault_Rest",
                       I_ManMode := "ManMode",
                       Q_AdvEnd => "变频器4正转到位(不用",
                       Q_RetEnd => "变频器4反转到位(不用",
                       O_AdvRot => #下线体正转,
                       O_RetRot => #下线体反转,
                       O_HiSpeed => #下线体高速,
                       O_LoSpeed => #下线体低速,
                       O_InvRes => #下线体复位);
   "前段_INV4正转" := #下线体正转;
   "后段_INV6正转" := #下线体正转;
   "前段_INV4速度1" := #下线体高速;
   "后段_INV6速度1" := #下线体高速;
   "前段_INV4速度2" := #下线体低速;
   "后段_INV6速度2" := #下线体低速;
   "前段_INV4复位" := #下线体复位;
   "后段_INV6复位" := #下线体复位;
END_REGION
END_FUNCTION_BLOCK

FUNCTION_BLOCK "F100_Val"   // FB100, LAD
TITLE = 电磁阀控制，
{ S7_Optimized_Access := 'TRUE' }
VERSION : 0.1
// IW_ConMode    00= 双端实际传感器到位，10=出端虚拟到位，11=出双端虚拟到位，01=回端端虚拟到位，
// stored: AutoNumber false, IsIECCheckEnabled false, IsRetainMemResEnabled false, MemoryReserve 100, SetENOAutomatically false, UDAEnableTagReadback false
   VAR_INPUT
      I_AutoAdv : Bool;   // 自动出指令
      I_AutoRet : Bool;   // 自动回指令
      I_ManAdv : Bool;   // 手动出指令
      I_ManRet : Bool;   // 手动回指令
      I_AdvCond : Bool;   // 动作出条件
      I_RetCond : Bool;   // 动作回条件
      I_AdvLS : Bool;   // 伸出到位
      I_RetLS : Bool;   // 返回到位
      IW_AdvTime : Time;   // 出or虚拟延迟
      IW_RetTime : Time;   // 回or虚拟延迟
      IW_AdvTimeOver : Time;   // 伸出超时
      IW_RetTimeOver : Time;   // 返回超时
      I_FoBrRel : Bool;   // 刹车强制解除
      I_Rest : Bool;   // 异常复位
      I_ManMode : Bool;   // 手动模式
      IW_ConMode : UInt;   // 虚拟控制
   END_VAR
   VAR_OUTPUT
      Q_AdvEnd : Bool;   // 伸出到位延迟
      Q_RetEnd : Bool;   // 返回到位延迟
      Q_AdvLS : Bool;   // 伸出到位
      Q_RetLS : Bool;   // 返回到位
      Q_AdvSL : Bool;   // 伸出输出
      Q_RetSL : Bool;   // 返回输出
      Q_FoBraRel : Bool;   // 刹车解除输出
      Q_AdvTiOvErr { ExternalAccessible := 'False'; ExternalVisible := 'False'; ExternalWritable := 'False'} : Bool;   // 出动作超时故障
      Q_RetTiOvErr { ExternalAccessible := 'False'; ExternalVisible := 'False'; ExternalWritable := 'False'} : Bool;   // 回动作超时故障
      Q_SensorsErr : Bool;   // 到位传感器都ON故障
      Q_SenCroErr : Bool;   // 到位传感器交叉ON故障
   END_VAR
   VAR
      MT_AdvChK { ExternalAccessible := 'False'; ExternalVisible := 'False'; ExternalWritable := 'False'} : IEC_TIMER;   // 出端延迟
      MT_RetChK { ExternalAccessible := 'False'; ExternalVisible := 'False'; ExternalWritable := 'False'} : IEC_TIMER;   // 回端延迟
      MT_AdvChKVir { ExternalAccessible := 'False'; ExternalVisible := 'False'; ExternalWritable := 'False'} : IEC_TIMER;   // 出端虚拟延迟
      MT_RetChKVir { ExternalAccessible := 'False'; ExternalVisible := 'False'; ExternalWritable := 'False'} : IEC_TIMER;   // 回端虚拟延迟
      MT_AdvTimeOver { ExternalAccessible := 'False'; ExternalVisible := 'False'; ExternalWritable := 'False'} : IEC_TIMER;   // 出动作延迟
      MT_RetTimeOver { ExternalAccessible := 'False'; ExternalVisible := 'False'; ExternalWritable := 'False'} : IEC_TIMER;   // 回动作延迟
   END_VAR
   VAR_TEMP
      M_AdvComm : Bool;   // 出动作
      M_RetComm : Bool;   // 回动作
      M_AdvM : Bool;   // 出指令
      M_RetM : Bool;   // 回指令
      M_SensorsErr : Bool;   // 到位传感器都ON
      M_SenCroErr : Bool;   // 到位传感器交叉ON
   END_VAR
   VAR_TEMP   // added for the SCL form of the ladder/FBD networks
      _w1 : Bool;
   END_VAR
BEGIN

REGION Network 1: 控制指令
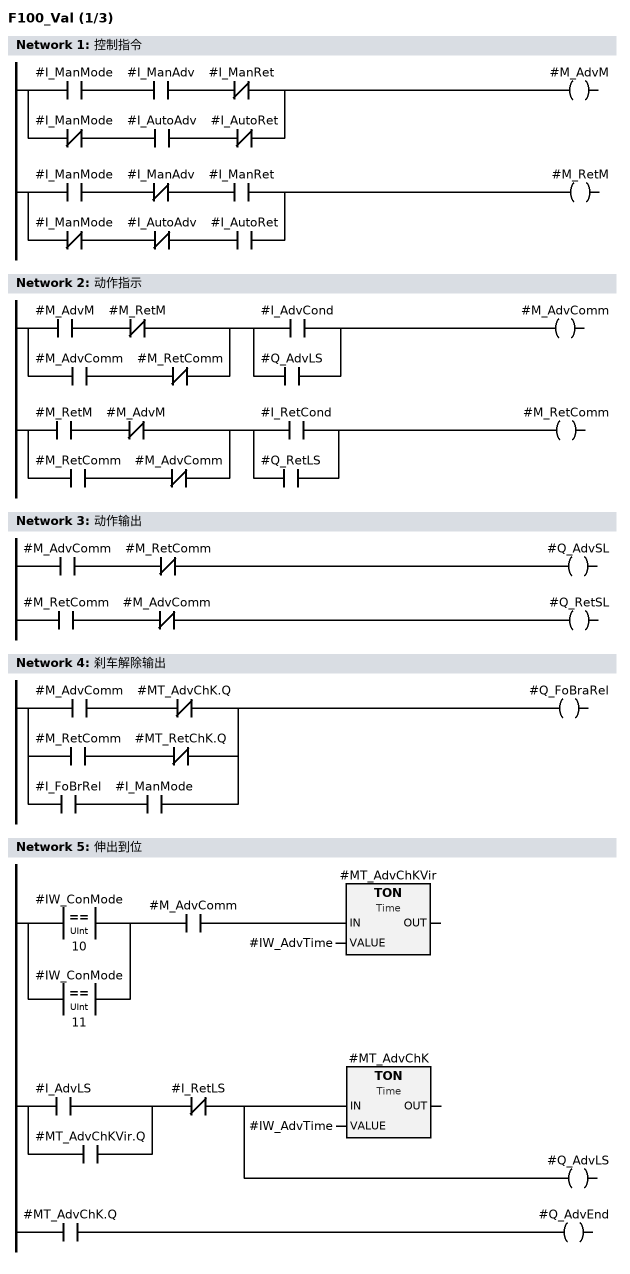
   RUNG wire#powerrail
      Contact( #I_ManMode )
      Contact( #I_ManAdv )
      I_Contact( #I_ManRet )
      wire#w1
      Coil( #M_AdvM )
   END_RUNG
   RUNG wire#powerrail
      I_Contact( #I_ManMode )
      Contact( #I_AutoAdv )
      I_Contact( #I_AutoRet )
   END_RUNG wire#w1
   RUNG wire#powerrail
      Contact( #I_ManMode )
      I_Contact( #I_ManAdv )
      Contact( #I_ManRet )
      wire#w2
      Coil( #M_RetM )
   END_RUNG
   RUNG wire#powerrail
      I_Contact( #I_ManMode )
      I_Contact( #I_AutoAdv )
      Contact( #I_AutoRet )
   END_RUNG wire#w2
   // the same network as SCL:
   #M_AdvM := (#I_ManMode AND #I_ManAdv AND NOT #I_ManRet) OR (NOT #I_ManMode AND #I_AutoAdv AND NOT #I_AutoRet);
   #M_RetM := (#I_ManMode AND NOT #I_ManAdv AND #I_ManRet) OR (NOT #I_ManMode AND NOT #I_AutoAdv AND #I_AutoRet);
END_REGION

REGION Network 2: 动作指示
   RUNG wire#powerrail
      Contact( #M_AdvM )
      I_Contact( #M_RetM )
      wire#w1
      Contact( #I_AdvCond )
      wire#w2
      Coil( #M_AdvComm )
   END_RUNG
   RUNG wire#powerrail
      Contact( #M_AdvComm )
      I_Contact( #M_RetComm )
   END_RUNG wire#w1
   RUNG wire#w1
      Contact( #Q_AdvLS )
   END_RUNG wire#w2
   RUNG wire#powerrail
      Contact( #M_RetM )
      I_Contact( #M_AdvM )
      wire#w3
      Contact( #I_RetCond )
      wire#w4
      Coil( #M_RetComm )
   END_RUNG
   RUNG wire#powerrail
      Contact( #M_RetComm )
      I_Contact( #M_AdvComm )
   END_RUNG wire#w3
   RUNG wire#w3
      Contact( #Q_RetLS )
   END_RUNG wire#w4
   // the same network as SCL:
   #M_AdvComm := ((#M_AdvM AND NOT #M_RetM) OR (#M_AdvComm AND NOT #M_RetComm)) AND (#I_AdvCond OR #Q_AdvLS);
   #M_RetComm := ((#M_RetM AND NOT #M_AdvM) OR (#M_RetComm AND NOT #M_AdvComm)) AND (#I_RetCond OR #Q_RetLS);
END_REGION

REGION Network 3: 动作输出
   RUNG wire#powerrail
      Contact( #M_AdvComm )
      I_Contact( #M_RetComm )
      Coil( #Q_AdvSL )
   END_RUNG
   RUNG wire#powerrail
      Contact( #M_RetComm )
      I_Contact( #M_AdvComm )
      Coil( #Q_RetSL )
   END_RUNG
   // the same network as SCL:
   #Q_AdvSL := #M_AdvComm AND NOT #M_RetComm;
   #Q_RetSL := #M_RetComm AND NOT #M_AdvComm;
END_REGION

REGION Network 4: 刹车解除输出
   RUNG wire#powerrail
      Contact( #M_AdvComm )
      I_Contact( #MT_AdvChK.Q )
      wire#w1
      Coil( #Q_FoBraRel )
   END_RUNG
   RUNG wire#powerrail
      Contact( #M_RetComm )
      I_Contact( #MT_RetChK.Q )
   END_RUNG wire#w1
   RUNG wire#powerrail
      Contact( #I_FoBrRel )
      Contact( #I_ManMode )
   END_RUNG wire#w1
   // the same network as SCL:
   #Q_FoBraRel := (#M_AdvComm AND NOT #MT_AdvChK.Q) OR (#M_RetComm AND NOT #MT_RetChK.Q) OR (#I_FoBrRel AND #I_ManMode);
END_REGION

REGION Network 5: 伸出到位
   #MT_AdvChKVir.TON(IN := ((#IW_ConMode = 10) OR (#IW_ConMode = 11)) AND #M_AdvComm, PT := #IW_AdvTime);   // TON coil
   #_w1 := (#I_AdvLS OR #MT_AdvChKVir.Q) AND NOT #I_RetLS;
   #MT_AdvChK.TON(IN := #_w1, PT := #IW_AdvTime);   // TON coil
   #Q_AdvLS := #_w1;
   #Q_AdvEnd := #MT_AdvChK.Q;
END_REGION

REGION Network 6: 返回到位
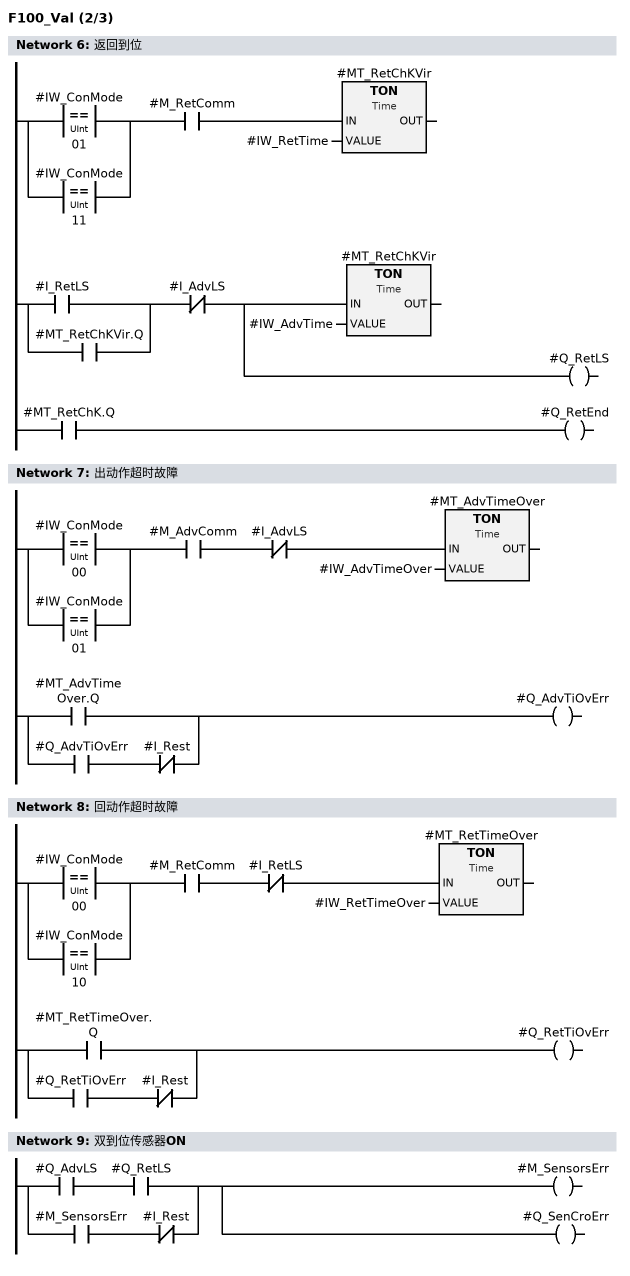
   #MT_RetChKVir.TON(IN := ((#IW_ConMode = 01) OR (#IW_ConMode = 11)) AND #M_RetComm, PT := #IW_RetTime);   // TON coil
   #_w1 := (#I_RetLS OR #MT_RetChKVir.Q) AND NOT #I_AdvLS;
   #MT_RetChKVir.TON(IN := #_w1, PT := #IW_AdvTime);   // TON coil
   #Q_RetLS := #_w1;
   #Q_RetEnd := #MT_RetChK.Q;
END_REGION

REGION Network 7: 出动作超时故障
   #MT_AdvTimeOver.TON(IN := ((#IW_ConMode = 00) OR (#IW_ConMode = 01)) AND #M_AdvComm AND NOT #I_AdvLS, PT := #IW_AdvTimeOver);   // TON coil
   #Q_AdvTiOvErr := #MT_AdvTimeOver.Q OR (#Q_AdvTiOvErr AND NOT #I_Rest);
END_REGION

REGION Network 8: 回动作超时故障
   #MT_RetTimeOver.TON(IN := ((#IW_ConMode = 00) OR (#IW_ConMode = 10)) AND #M_RetComm AND NOT #I_RetLS, PT := #IW_RetTimeOver);   // TON coil
   #Q_RetTiOvErr := #MT_RetTimeOver.Q OR (#Q_RetTiOvErr AND NOT #I_Rest);
END_REGION

REGION Network 9: 双到位传感器ON
   RUNG wire#powerrail
      Contact( #Q_AdvLS )
      Contact( #Q_RetLS )
      wire#w1
      Coil( #M_SensorsErr )
   END_RUNG
   RUNG wire#powerrail
      Contact( #M_SensorsErr )
      I_Contact( #I_Rest )
   END_RUNG wire#w1
   RUNG wire#w1
      Coil( #Q_SenCroErr )
   END_RUNG
   // the same network as SCL:
   #M_SensorsErr := (#Q_AdvLS AND #Q_RetLS) OR (#M_SensorsErr AND NOT #I_Rest);
   #Q_SenCroErr := #M_SensorsErr;
END_REGION

REGION Network 10: 到位传感器交叉ON
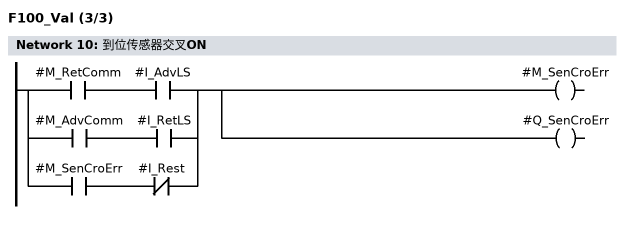
   RUNG wire#powerrail
      Contact( #M_RetComm )
      Contact( #I_AdvLS )
      wire#w1
      Coil( #M_SenCroErr )
   END_RUNG
   RUNG wire#powerrail
      Contact( #M_AdvComm )
      Contact( #I_RetLS )
   END_RUNG wire#w1
   RUNG wire#powerrail
      Contact( #M_SenCroErr )
      I_Contact( #I_Rest )
   END_RUNG wire#w1
   RUNG wire#w1
      Coil( #Q_SenCroErr )
   END_RUNG
   // the same network as SCL:
   #M_SenCroErr := (#M_RetComm AND #I_AdvLS) OR (#M_AdvComm AND #I_RetLS) OR (#M_SenCroErr AND NOT #I_Rest);
   #Q_SenCroErr := #M_SenCroErr;
END_REGION
END_FUNCTION_BLOCK

FUNCTION_BLOCK "F110_Inv"   // FB110, LAD
{ S7_Optimized_Access := 'TRUE' }
VERSION : 0.1
// 变频器FB
// stored: AutoNumber false, IsIECCheckEnabled false, IsRetainMemResEnabled false, MemoryReserve 100, SetENOAutomatically false, UDAEnableTagReadback false
   VAR_INPUT
      I_AutoAdv : Bool;   // 自动正转指令
      I_AutoRet : Bool;   // 自动反转指令
      I_ManAdv : Bool;   // 手动正转指令
      I_ManRet : Bool;   // 手动反转指令
      I_AdvCond : Bool;   // 正转动作条件
      I_RetCond : Bool;   // 反转动作条件
      I_AdvLS : Bool;   // 正转到位
      I_RetLS : Bool;   // 反转到位
      I_AdLowP : Bool;   // 正转减速位置
      I_ReLowP : Bool;   // 反转减速位置
      I_InvNorm : Bool;   // 变频器正常
      I_InvCut : Bool;   // 变频器切断
      IW_ChkTim : Time;   // 动作确认时间
      I_FoBrRel : Bool;   // 刹车强制解除
      I_Rest : Bool;   // 异常复位
      I_ManMode : Bool;   // 手动模式
   END_VAR
   VAR_OUTPUT
      Q_AdvEnd : Bool;   // 正转到位
      Q_RetEnd : Bool;   // 反转到位
      O_AdvRot : Bool;   // 正转
      O_RetRot : Bool;   // 反转
      O_HiSpeed : Bool;   // 高速
      O_LoSpeed { ExternalVisible := 'False'} : Bool;   // 低速
      O_InvRes : Bool;   // INV.复位输出
      O_InvStop : Bool;   // INV.输出正常
      O_BrRel : Bool;   // 制动器解除输出
      O_LS_Flt : Bool;   // LS异常
      O_ActFlt : Bool;   // 动作异常
      O_InvFlt : Bool;   // 变频器异常
   END_VAR
   VAR
      MT_ActF : IEC_TIMER;   // 动作异常
   END_VAR
   VAR_TEMP
      M_MoveOK : Bool;   // 动作可
      M_AdvM : Bool;   // 正转操作
      M_RetM : Bool;   // 反转操作
      M_AdvComm : Bool;   // 正转指示
      M_RetComm : Bool;   // 反转指示
      M_TimOf : Bool;   // 动作无效确认
   END_VAR
   VAR_TEMP   // added for the SCL form of the ladder/FBD networks
      _w1 : Bool;
   END_VAR
BEGIN

REGION Network 1: 动作无效确认
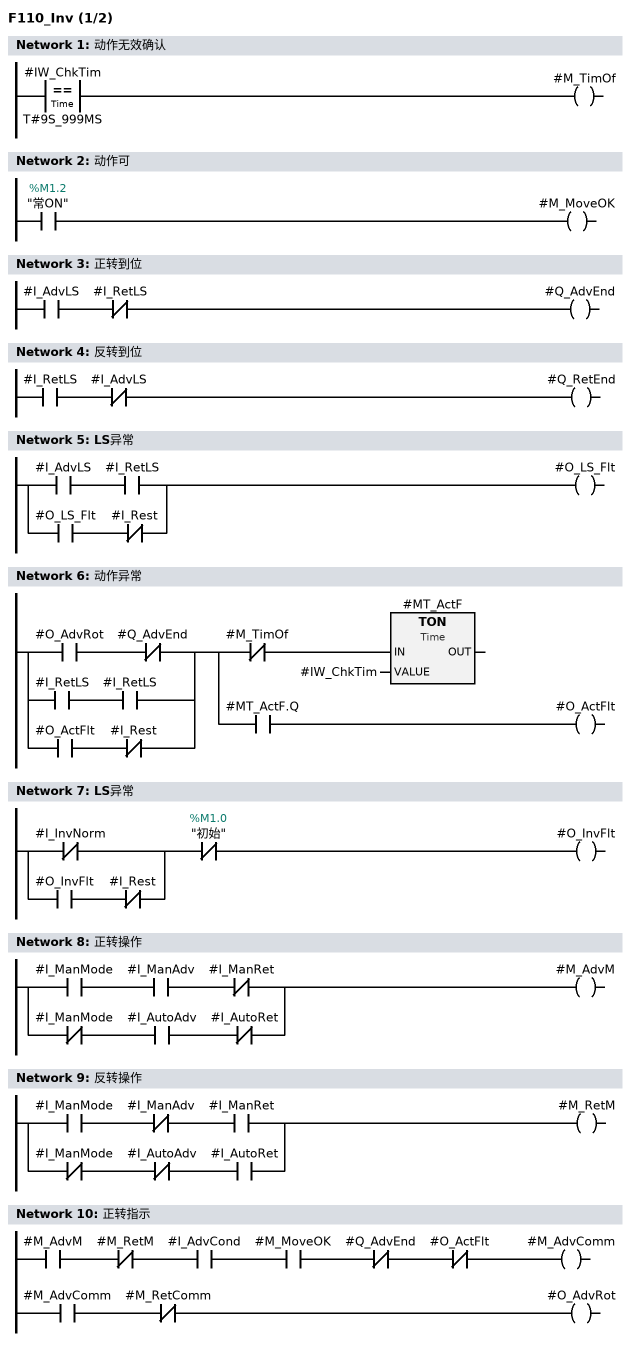
   RUNG wire#powerrail
      { S7_Templates := "SrcType := Time" } EQ_Contact(in1 := #IW_ChkTim, in2 := T#9S_999MS)
      Coil( #M_TimOf )
   END_RUNG
   // the same network as SCL:
   #M_TimOf := #IW_ChkTim = T#9S_999MS;
END_REGION

REGION Network 2: 动作可
   RUNG wire#powerrail
      Contact( "常ON" )
      Coil( #M_MoveOK )
   END_RUNG
   // the same network as SCL:
   #M_MoveOK := "常ON";
END_REGION

REGION Network 3: 正转到位
   RUNG wire#powerrail
      Contact( #I_AdvLS )
      I_Contact( #I_RetLS )
      Coil( #Q_AdvEnd )
   END_RUNG
   // the same network as SCL:
   #Q_AdvEnd := #I_AdvLS AND NOT #I_RetLS;
END_REGION

REGION Network 4: 反转到位
   RUNG wire#powerrail
      Contact( #I_RetLS )
      I_Contact( #I_AdvLS )
      Coil( #Q_RetEnd )
   END_RUNG
   // the same network as SCL:
   #Q_RetEnd := #I_RetLS AND NOT #I_AdvLS;
END_REGION

REGION Network 5: LS异常
   RUNG wire#powerrail
      Contact( #I_AdvLS )
      Contact( #I_RetLS )
      wire#w1
      Coil( #O_LS_Flt )
   END_RUNG
   RUNG wire#powerrail
      Contact( #O_LS_Flt )
      I_Contact( #I_Rest )
   END_RUNG wire#w1
   // the same network as SCL:
   #O_LS_Flt := (#I_AdvLS AND #I_RetLS) OR (#O_LS_Flt AND NOT #I_Rest);
END_REGION

REGION Network 6: 动作异常
   #_w1 := (#O_AdvRot AND NOT #Q_AdvEnd) OR (#I_RetLS AND #I_RetLS) OR (#O_ActFlt AND NOT #I_Rest);
   #MT_ActF.TON(IN := #_w1 AND NOT #M_TimOf, PT := #IW_ChkTim);   // TON coil
   #O_ActFlt := #_w1 AND #MT_ActF.Q;
END_REGION

REGION Network 7: LS异常
   RUNG wire#powerrail
      I_Contact( #I_InvNorm )
      wire#w1
      I_Contact( "初始" )
      Coil( #O_InvFlt )
   END_RUNG
   RUNG wire#powerrail
      Contact( #O_InvFlt )
      I_Contact( #I_Rest )
   END_RUNG wire#w1
   // the same network as SCL:
   #O_InvFlt := (NOT #I_InvNorm OR (#O_InvFlt AND NOT #I_Rest)) AND NOT "初始";
END_REGION

REGION Network 8: 正转操作
   RUNG wire#powerrail
      Contact( #I_ManMode )
      Contact( #I_ManAdv )
      I_Contact( #I_ManRet )
      wire#w1
      Coil( #M_AdvM )
   END_RUNG
   RUNG wire#powerrail
      I_Contact( #I_ManMode )
      Contact( #I_AutoAdv )
      I_Contact( #I_AutoRet )
   END_RUNG wire#w1
   // the same network as SCL:
   #M_AdvM := (#I_ManMode AND #I_ManAdv AND NOT #I_ManRet) OR (NOT #I_ManMode AND #I_AutoAdv AND NOT #I_AutoRet);
END_REGION

REGION Network 9: 反转操作
   RUNG wire#powerrail
      Contact( #I_ManMode )
      I_Contact( #I_ManAdv )
      Contact( #I_ManRet )
      wire#w1
      Coil( #M_RetM )
   END_RUNG
   RUNG wire#powerrail
      I_Contact( #I_ManMode )
      I_Contact( #I_AutoAdv )
      Contact( #I_AutoRet )
   END_RUNG wire#w1
   // the same network as SCL:
   #M_RetM := (#I_ManMode AND NOT #I_ManAdv AND #I_ManRet) OR (NOT #I_ManMode AND NOT #I_AutoAdv AND #I_AutoRet);
END_REGION

REGION Network 10: 正转指示
   RUNG wire#powerrail
      Contact( #M_AdvM )
      I_Contact( #M_RetM )
      Contact( #I_AdvCond )
      Contact( #M_MoveOK )
      I_Contact( #Q_AdvEnd )
      I_Contact( #O_ActFlt )
      Coil( #M_AdvComm )
   END_RUNG
   RUNG wire#powerrail
      Contact( #M_AdvComm )
      I_Contact( #M_RetComm )
      Coil( #O_AdvRot )
   END_RUNG
   // the same network as SCL:
   #M_AdvComm := #M_AdvM AND NOT #M_RetM AND #I_AdvCond AND #M_MoveOK AND NOT #Q_AdvEnd AND NOT #O_ActFlt;
   #O_AdvRot := #M_AdvComm AND NOT #M_RetComm;
END_REGION

REGION Network 11: 反转指示
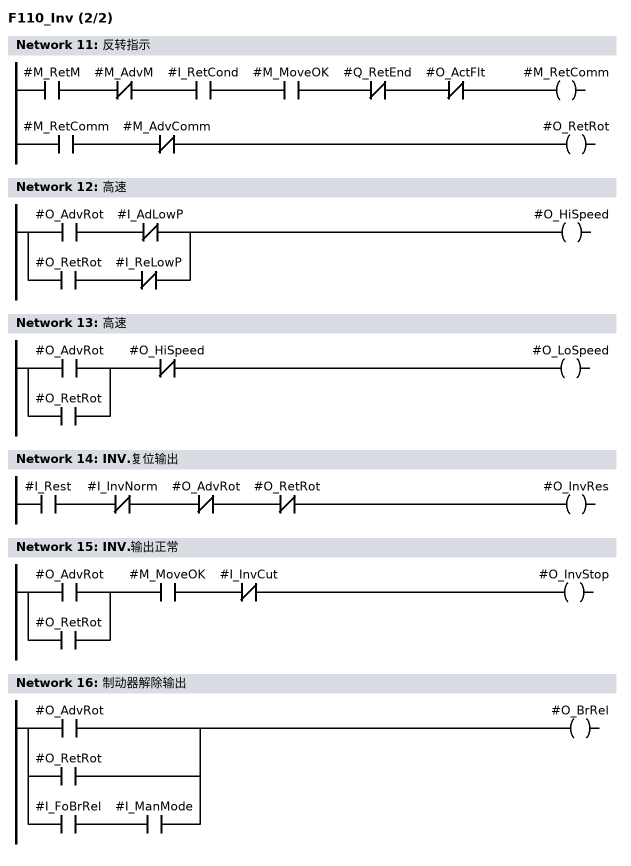
   RUNG wire#powerrail
      Contact( #M_RetM )
      I_Contact( #M_AdvM )
      Contact( #I_RetCond )
      Contact( #M_MoveOK )
      I_Contact( #Q_RetEnd )
      I_Contact( #O_ActFlt )
      Coil( #M_RetComm )
   END_RUNG
   RUNG wire#powerrail
      Contact( #M_RetComm )
      I_Contact( #M_AdvComm )
      Coil( #O_RetRot )
   END_RUNG
   // the same network as SCL:
   #M_RetComm := #M_RetM AND NOT #M_AdvM AND #I_RetCond AND #M_MoveOK AND NOT #Q_RetEnd AND NOT #O_ActFlt;
   #O_RetRot := #M_RetComm AND NOT #M_AdvComm;
END_REGION

REGION Network 12: 高速
   RUNG wire#powerrail
      Contact( #O_AdvRot )
      I_Contact( #I_AdLowP )
      wire#w1
      Coil( #O_HiSpeed )
   END_RUNG
   RUNG wire#powerrail
      Contact( #O_RetRot )
      I_Contact( #I_ReLowP )
   END_RUNG wire#w1
   // the same network as SCL:
   #O_HiSpeed := (#O_AdvRot AND NOT #I_AdLowP) OR (#O_RetRot AND NOT #I_ReLowP);
END_REGION

REGION Network 13: 高速
   RUNG wire#powerrail
      Contact( #O_AdvRot )
      wire#w1
      I_Contact( #O_HiSpeed )
      Coil( #O_LoSpeed )
   END_RUNG
   RUNG wire#powerrail
      Contact( #O_RetRot )
   END_RUNG wire#w1
   // the same network as SCL:
   #O_LoSpeed := (#O_AdvRot OR #O_RetRot) AND NOT #O_HiSpeed;
END_REGION

REGION Network 14: INV.复位输出
   RUNG wire#powerrail
      Contact( #I_Rest )
      I_Contact( #I_InvNorm )
      I_Contact( #O_AdvRot )
      I_Contact( #O_RetRot )
      Coil( #O_InvRes )
   END_RUNG
   // the same network as SCL:
   #O_InvRes := #I_Rest AND NOT #I_InvNorm AND NOT #O_AdvRot AND NOT #O_RetRot;
END_REGION

REGION Network 15: INV.输出正常
   RUNG wire#powerrail
      Contact( #O_AdvRot )
      wire#w1
      Contact( #M_MoveOK )
      I_Contact( #I_InvCut )
      Coil( #O_InvStop )
   END_RUNG
   RUNG wire#powerrail
      Contact( #O_RetRot )
   END_RUNG wire#w1
   // the same network as SCL:
   #O_InvStop := (#O_AdvRot OR #O_RetRot) AND #M_MoveOK AND NOT #I_InvCut;
END_REGION

REGION Network 16: 制动器解除输出
   RUNG wire#powerrail
      Contact( #O_AdvRot )
      wire#w1
      Coil( #O_BrRel )
   END_RUNG
   RUNG wire#powerrail
      Contact( #O_RetRot )
   END_RUNG wire#w1
   RUNG wire#powerrail
      Contact( #I_FoBrRel )
      Contact( #I_ManMode )
   END_RUNG wire#w1
   // the same network as SCL:
   #O_BrRel := #O_AdvRot OR #O_RetRot OR (#I_FoBrRel AND #I_ManMode);
END_REGION
END_FUNCTION_BLOCK

FUNCTION_BLOCK "K07_轴组"   // FB7, LAD
{ S7_Optimized_Access := 'TRUE' }
VERSION : 0.1
// stored: AutoNumber false, IsIECCheckEnabled false, IsRetainMemResEnabled false, MemoryReserve 100, SetENOAutomatically false, UDAEnableTagReadback false
   VAR
      Axis1Write { S7_SetPoint := 'True'} : "F121_SinaParaWrite(SV660F)";   // 轴1参数
      Axis1Pos { S7_SetPoint := 'True'} : "F120_SinaPos(SV660F)";   // 轴1定位
   END_VAR
   VAR_TEMP   // added for the SCL form of the ladder/FBD networks
      _w1 : Bool;
      _w2 : Bool;
      _w3 : Bool;
      _w4 : Bool;
      _w5 : Bool;
      _w6 : Bool;
      _w7 : Bool;
      _w8 : Bool;
      _w9 : Bool;
   END_VAR
BEGIN

REGION Network 1: 轴1参数
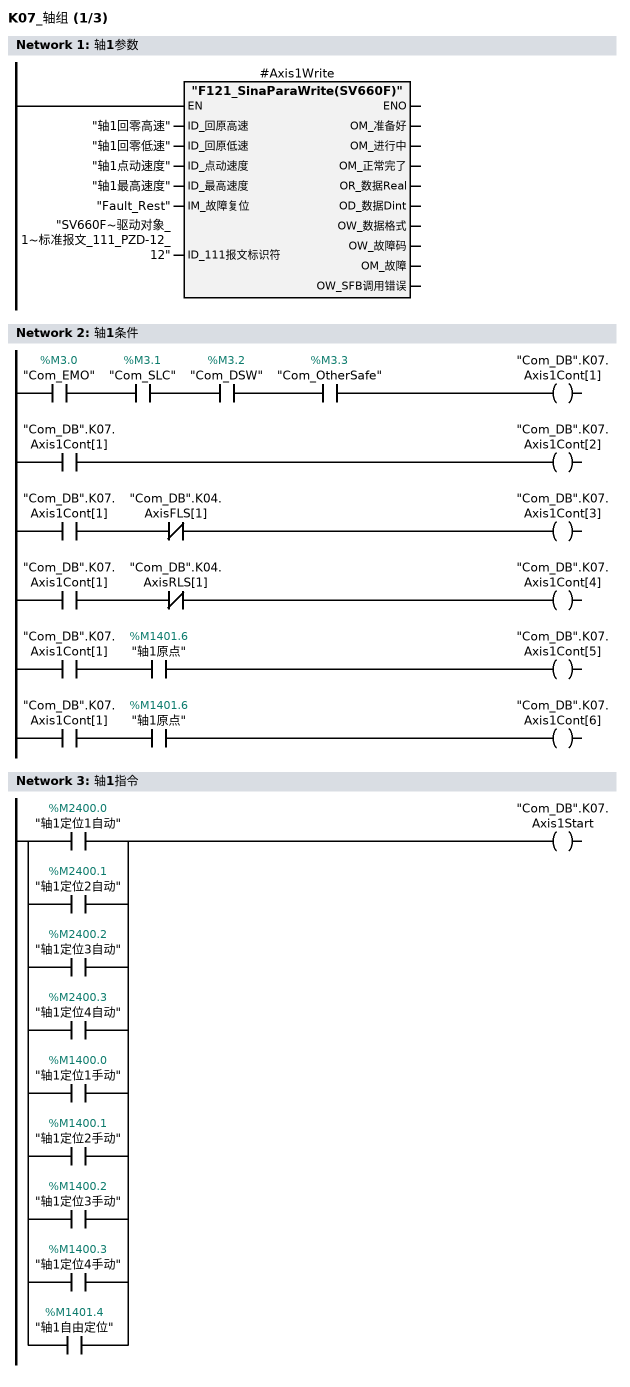
   RUNG wire#powerrail
      #Axis1Write(ID_回原高速 := "轴1回零高速", ID_回原低速 := "轴1回零低速", ID_点动速度 := "轴1点动速度", ID_最高速度 := "轴1最高速度", IM_故障复位 := "Fault_Rest", ID_111报文标识符 := "SV660F~驱动对象_1~标准报文_111_PZD-12_12", OM_准备好 =>, OM_进行中 =>, OM_正常完了 =>, OR_数据Real =>, OD_数据Dint =>, OW_数据格式 =>, OW_故障码 =>, OM_故障 =>, OW_SFB调用错误 =>)
   END_RUNG
   // the same network as SCL:
   #Axis1Write(ID_回原高速 := "轴1回零高速",   // "F121_SinaParaWrite(SV660F)"
               ID_回原低速 := "轴1回零低速",
               ID_点动速度 := "轴1点动速度",
               ID_最高速度 := "轴1最高速度",
               IM_故障复位 := "Fault_Rest",
               ID_111报文标识符 := "SV660F~驱动对象_1~标准报文_111_PZD-12_12");
END_REGION

REGION Network 2: 轴1条件
   RUNG wire#powerrail
      Contact( "Com_EMO" )
      Contact( "Com_SLC" )
      Contact( "Com_DSW" )
      Contact( "Com_OtherSafe" )
      Coil( "Com_DB".K07.Axis1Cont[1] )
   END_RUNG
   RUNG wire#powerrail
      Contact( "Com_DB".K07.Axis1Cont[1] )
      Coil( "Com_DB".K07.Axis1Cont[2] )
   END_RUNG
   RUNG wire#powerrail
      Contact( "Com_DB".K07.Axis1Cont[1] )
      I_Contact( "Com_DB".K04.AxisFLS[1] )
      Coil( "Com_DB".K07.Axis1Cont[3] )
   END_RUNG
   RUNG wire#powerrail
      Contact( "Com_DB".K07.Axis1Cont[1] )
      I_Contact( "Com_DB".K04.AxisRLS[1] )
      Coil( "Com_DB".K07.Axis1Cont[4] )
   END_RUNG
   RUNG wire#powerrail
      Contact( "Com_DB".K07.Axis1Cont[1] )
      Contact( "轴1原点" )
      Coil( "Com_DB".K07.Axis1Cont[5] )
   END_RUNG
   RUNG wire#powerrail
      Contact( "Com_DB".K07.Axis1Cont[1] )
      Contact( "轴1原点" )
      Coil( "Com_DB".K07.Axis1Cont[6] )
   END_RUNG
   // the same network as SCL:
   "Com_DB".K07.Axis1Cont[1] := "Com_EMO" AND "Com_SLC" AND "Com_DSW" AND "Com_OtherSafe";
   "Com_DB".K07.Axis1Cont[2] := "Com_DB".K07.Axis1Cont[1];
   "Com_DB".K07.Axis1Cont[3] := "Com_DB".K07.Axis1Cont[1] AND NOT "Com_DB".K04.AxisFLS[1];
   "Com_DB".K07.Axis1Cont[4] := "Com_DB".K07.Axis1Cont[1] AND NOT "Com_DB".K04.AxisRLS[1];
   "Com_DB".K07.Axis1Cont[5] := "Com_DB".K07.Axis1Cont[1] AND "轴1原点";
   "Com_DB".K07.Axis1Cont[6] := "Com_DB".K07.Axis1Cont[1] AND "轴1原点";
END_REGION

REGION Network 3: 轴1指令
   RUNG wire#powerrail
      Contact( "轴1定位1自动" )
      wire#w1
      Coil( "Com_DB".K07.Axis1Start )
   END_RUNG
   RUNG wire#powerrail
      Contact( "轴1定位2自动" )
   END_RUNG wire#w1
   RUNG wire#powerrail
      Contact( "轴1定位3自动" )
   END_RUNG wire#w1
   RUNG wire#powerrail
      Contact( "轴1定位4自动" )
   END_RUNG wire#w1
   RUNG wire#powerrail
      Contact( "轴1定位1手动" )
   END_RUNG wire#w1
   RUNG wire#powerrail
      Contact( "轴1定位2手动" )
   END_RUNG wire#w1
   RUNG wire#powerrail
      Contact( "轴1定位3手动" )
   END_RUNG wire#w1
   RUNG wire#powerrail
      Contact( "轴1定位4手动" )
   END_RUNG wire#w1
   RUNG wire#powerrail
      Contact( "轴1自由定位" )
   END_RUNG wire#w1
   // the same network as SCL:
   "Com_DB".K07.Axis1Start := "轴1定位1自动" OR "轴1定位2自动" OR "轴1定位3自动" OR "轴1定位4自动" OR "轴1定位1手动" OR "轴1定位2手动" OR "轴1定位3手动" OR "轴1定位4手动" OR "轴1自由定位";
END_REGION

REGION Network 4: 轴1位置速度
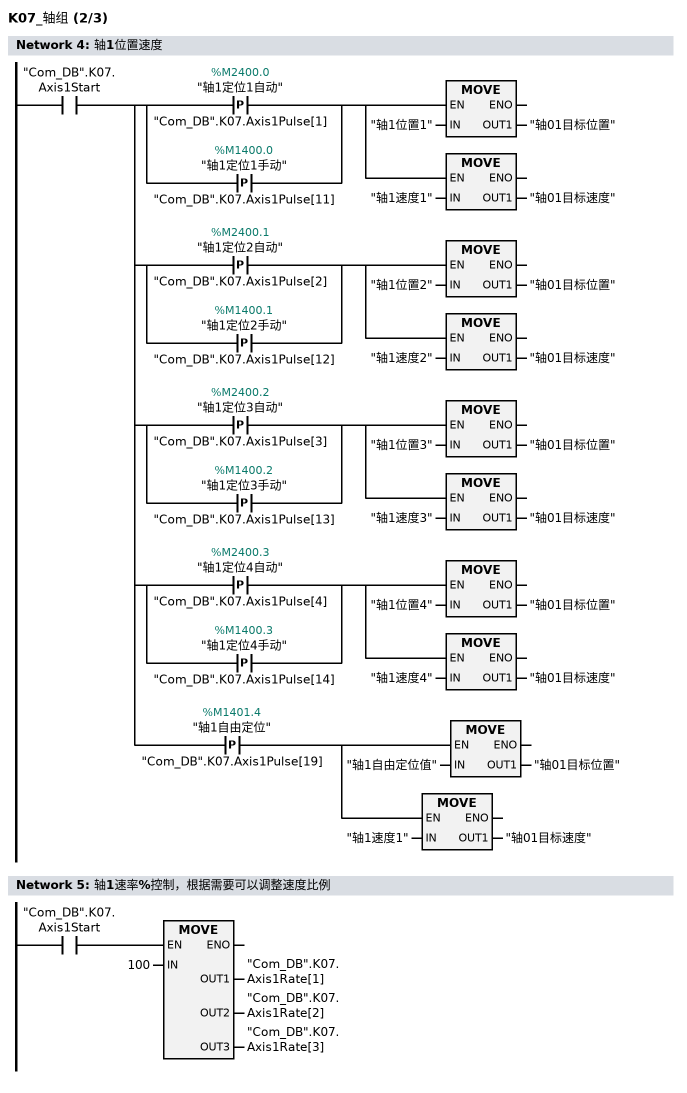
   RUNG wire#powerrail
      Contact( "Com_DB".K07.Axis1Start )
      wire#w1
      P_Contact(operand := "轴1定位1自动", bit := "Com_DB".K07.Axis1Pulse[1])
      wire#w2
      Move(in := "轴1位置1", out1 => "轴01目标位置")
   END_RUNG
   RUNG wire#w1
      P_Contact(operand := "轴1定位1手动", bit := "Com_DB".K07.Axis1Pulse[11])
   END_RUNG wire#w2
   RUNG wire#w2
      Move(in := "轴1速度1", out1 => "轴01目标速度")
   END_RUNG
   RUNG wire#w1
      P_Contact(operand := "轴1定位2自动", bit := "Com_DB".K07.Axis1Pulse[2])
      wire#w3
      Move(in := "轴1位置2", out1 => "轴01目标位置")
   END_RUNG
   RUNG wire#w1
      P_Contact(operand := "轴1定位2手动", bit := "Com_DB".K07.Axis1Pulse[12])
   END_RUNG wire#w3
   RUNG wire#w3
      Move(in := "轴1速度2", out1 => "轴01目标速度")
   END_RUNG
   RUNG wire#w1
      P_Contact(operand := "轴1定位3自动", bit := "Com_DB".K07.Axis1Pulse[3])
      wire#w4
      Move(in := "轴1位置3", out1 => "轴01目标位置")
   END_RUNG
   RUNG wire#w1
      P_Contact(operand := "轴1定位3手动", bit := "Com_DB".K07.Axis1Pulse[13])
   END_RUNG wire#w4
   RUNG wire#w4
      Move(in := "轴1速度3", out1 => "轴01目标速度")
   END_RUNG
   RUNG wire#w1
      P_Contact(operand := "轴1定位4自动", bit := "Com_DB".K07.Axis1Pulse[4])
      wire#w5
      Move(in := "轴1位置4", out1 => "轴01目标位置")
   END_RUNG
   RUNG wire#w1
      P_Contact(operand := "轴1定位4手动", bit := "Com_DB".K07.Axis1Pulse[14])
   END_RUNG wire#w5
   RUNG wire#w5
      Move(in := "轴1速度4", out1 => "轴01目标速度")
   END_RUNG
   RUNG wire#w1
      P_Contact(operand := "轴1自由定位", bit := "Com_DB".K07.Axis1Pulse[19])
      wire#w6
      Move(in := "轴1自由定位值", out1 => "轴01目标位置")
   END_RUNG
   RUNG wire#w6
      Move(in := "轴1速度1", out1 => "轴01目标速度")
   END_RUNG
   // the same network as SCL:
   #_w1 := "Com_DB".K07.Axis1Start AND "轴1定位1自动" AND NOT "Com_DB".K07.Axis1Pulse[1];   // rising edge of "轴1定位1自动"
   "Com_DB".K07.Axis1Pulse[1] := "轴1定位1自动";
   #_w2 := "Com_DB".K07.Axis1Start AND "轴1定位1手动" AND NOT "Com_DB".K07.Axis1Pulse[11];   // rising edge of "轴1定位1手动"
   "Com_DB".K07.Axis1Pulse[11] := "轴1定位1手动";
   IF #_w1 OR #_w2 THEN
       "轴01目标位置" := "轴1位置1";
       "轴01目标速度" := "轴1速度1";
   END_IF;
   #_w3 := "Com_DB".K07.Axis1Start AND "轴1定位2自动" AND NOT "Com_DB".K07.Axis1Pulse[2];   // rising edge of "轴1定位2自动"
   "Com_DB".K07.Axis1Pulse[2] := "轴1定位2自动";
   #_w4 := "Com_DB".K07.Axis1Start AND "轴1定位2手动" AND NOT "Com_DB".K07.Axis1Pulse[12];   // rising edge of "轴1定位2手动"
   "Com_DB".K07.Axis1Pulse[12] := "轴1定位2手动";
   IF #_w3 OR #_w4 THEN
       "轴01目标位置" := "轴1位置2";
       "轴01目标速度" := "轴1速度2";
   END_IF;
   #_w5 := "Com_DB".K07.Axis1Start AND "轴1定位3自动" AND NOT "Com_DB".K07.Axis1Pulse[3];   // rising edge of "轴1定位3自动"
   "Com_DB".K07.Axis1Pulse[3] := "轴1定位3自动";
   #_w6 := "Com_DB".K07.Axis1Start AND "轴1定位3手动" AND NOT "Com_DB".K07.Axis1Pulse[13];   // rising edge of "轴1定位3手动"
   "Com_DB".K07.Axis1Pulse[13] := "轴1定位3手动";
   IF #_w5 OR #_w6 THEN
       "轴01目标位置" := "轴1位置3";
       "轴01目标速度" := "轴1速度3";
   END_IF;
   #_w7 := "Com_DB".K07.Axis1Start AND "轴1定位4自动" AND NOT "Com_DB".K07.Axis1Pulse[4];   // rising edge of "轴1定位4自动"
   "Com_DB".K07.Axis1Pulse[4] := "轴1定位4自动";
   #_w8 := "Com_DB".K07.Axis1Start AND "轴1定位4手动" AND NOT "Com_DB".K07.Axis1Pulse[14];   // rising edge of "轴1定位4手动"
   "Com_DB".K07.Axis1Pulse[14] := "轴1定位4手动";
   IF #_w7 OR #_w8 THEN
       "轴01目标位置" := "轴1位置4";
       "轴01目标速度" := "轴1速度4";
   END_IF;
   #_w9 := "Com_DB".K07.Axis1Start AND "轴1自由定位" AND NOT "Com_DB".K07.Axis1Pulse[19];   // rising edge of "轴1自由定位"
   "Com_DB".K07.Axis1Pulse[19] := "轴1自由定位";
   IF #_w9 THEN
       "轴01目标位置" := "轴1自由定位值";
       "轴01目标速度" := "轴1速度1";
   END_IF;
END_REGION

REGION Network 5: 轴1速率%控制，根据需要可以调整速度比例
   RUNG wire#powerrail
      Contact( "Com_DB".K07.Axis1Start )
      Move(in := 100, out1 => "Com_DB".K07.Axis1Rate[1], out2 => "Com_DB".K07.Axis1Rate[2], out3 => "Com_DB".K07.Axis1Rate[3])
   END_RUNG
   // the same network as SCL:
   IF "Com_DB".K07.Axis1Start THEN
       "Com_DB".K07.Axis1Rate[1] := 100;
       "Com_DB".K07.Axis1Rate[2] := 100;
       "Com_DB".K07.Axis1Rate[3] := 100;
   END_IF;
END_REGION

REGION Network 6: 轴1Pos
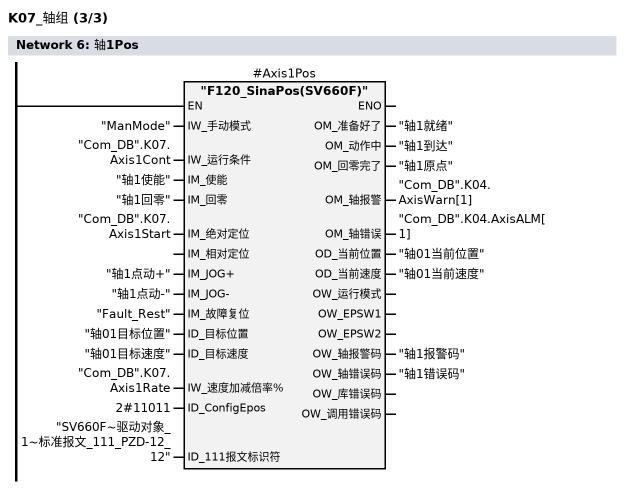
   RUNG wire#powerrail
      #Axis1Pos(IW_手动模式 := "ManMode", IW_运行条件 := "Com_DB".K07.Axis1Cont, IM_使能 := "轴1使能", IM_回零 := "轴1回零", IM_绝对定位 := "Com_DB".K07.Axis1Start, IM_相对定位 :=, "IM_JOG+" := "轴1点动+", "IM_JOG-" := "轴1点动-", IM_故障复位 := "Fault_Rest", ID_目标位置 := "轴01目标位置", ID_目标速度 := "轴01目标速度", "IW_速度加减倍率%" := "Com_DB".K07.Axis1Rate, ID_ConfigEpos := 2#11011, ID_111报文标识符 := "SV660F~驱动对象_1~标准报文_111_PZD-12_12", OM_准备好了 => "轴1就绪", OM_动作中 => "轴1到达", OM_回零完了 => "轴1原点", OM_轴报警 => "Com_DB".K04.AxisWarn[1], OM_轴错误 => "Com_DB".K04.AxisALM[1], OD_当前位置 => "轴01当前位置", OD_当前速度 => "轴01当前速度", OW_运行模式 =>, OW_EPSW1 =>, OW_EPSW2 =>, OW_轴报警码 => "轴1报警码", OW_轴错误码 => "轴1错误码", OW_库错误码 =>, OW_调用错误码 =>)
   END_RUNG
   // the same network as SCL:
   #Axis1Pos(IW_手动模式 := "ManMode",   // "F120_SinaPos(SV660F)"
             IW_运行条件 := "Com_DB".K07.Axis1Cont,
             IM_使能 := "轴1使能",
             IM_回零 := "轴1回零",
             IM_绝对定位 := "Com_DB".K07.Axis1Start,
             "IM_JOG+" := "轴1点动+",
             "IM_JOG-" := "轴1点动-",
             IM_故障复位 := "Fault_Rest",
             ID_目标位置 := "轴01目标位置",
             ID_目标速度 := "轴01目标速度",
             "IW_速度加减倍率%" := "Com_DB".K07.Axis1Rate,
             ID_ConfigEpos := 2#11011,
             ID_111报文标识符 := "SV660F~驱动对象_1~标准报文_111_PZD-12_12",
             OM_准备好了 => "轴1就绪",
             OM_动作中 => "轴1到达",
             OM_回零完了 => "轴1原点",
             OM_轴报警 => "Com_DB".K04.AxisWarn[1],
             OM_轴错误 => "Com_DB".K04.AxisALM[1],
             OD_当前位置 => "轴01当前位置",
             OD_当前速度 => "轴01当前速度",
             OW_轴报警码 => "轴1报警码",
             OW_轴错误码 => "轴1错误码");
END_REGION

REGION Network 7 (SCL): 轴1位置
   IF  ("轴1位置1"-2)<="轴01当前位置"
       AND ("轴1位置1"+2)>= "轴01当前位置"

   THEN
       "轴1定位1到位"           := TRUE         ;
   ELSE
       "轴1定位1到位" := FALSE;
   END_IF;// 

   IF ("轴1位置2" - 2) <= "轴01当前位置"
       AND ("轴1位置2" + 2) >= "轴01当前位置"

   THEN
       "轴1定位2到位" := TRUE;
   ELSE
       "轴1定位2到位" := FALSE;
   END_IF;

   IF ("轴1位置3" - 2) <= "轴01当前位置"
       AND ("轴1位置3" + 2) >= "轴01当前位置"

   THEN
       "轴1定位3到位" := TRUE;
   ELSE
       "轴1定位3到位" := FALSE;
   END_IF;

   IF ("轴1位置4" - 2) <= "轴01当前位置"
       AND ("轴1位置4" + 2) >= "轴01当前位置"

   THEN
       "轴1定位4到位" := TRUE;
   ELSE
       "轴1定位4到位" := FALSE;
   END_IF;
END_REGION

REGION Network 8: 轴1END
END_REGION
END_FUNCTION_BLOCK

FUNCTION_BLOCK "F121_SinaParaWrite(SV660F)"   // FB121, LAD
{ S7_Optimized_Access := 'TRUE' }
VERSION : 0.1
// stored: AutoNumber false, IsIECCheckEnabled false, IsRetainMemResEnabled false, MemoryReserve 100, SetENOAutomatically false, UDAEnableTagReadback false
   VAR_INPUT
      ID_回原高速 : DInt;
      ID_回原低速 : DInt;
      ID_点动速度 : DInt;
      ID_最高速度 : DInt;
      IM_故障复位 : Bool;
      ID_111报文标识符 { ExternalAccessible := 'False'; ExternalVisible := 'False'; ExternalWritable := 'False'} : HW_IO;
   END_VAR
   VAR_OUTPUT
      OM_准备好 : Bool;
      OM_进行中 : Bool;
      OM_正常完了 : Bool;
      OR_数据Real : Real;
      OD_数据Dint : DInt;
      OW_数据格式 : Int;
      OW_故障码 : Int;
      OM_故障 : Bool;
      OW_SFB调用错误 : Word;
   END_VAR
   VAR
      MT_Time { ExternalAccessible := 'False'; ExternalVisible := 'False'; ExternalWritable := 'False'} : IEC_TIMER;
   END_VAR
   VAR_TEMP
      MD_回原高速 : Array[1..2] of DInt;
      MD_回原低速 : Array[1..2] of DInt;
      MD_点动正速度 : Array[1..2] of DInt;
      MD_点动负速度 : Array[1..2] of DInt;
      MD_最高速度 : Array[1..2] of DInt;
      M_回原高速变更 : Bool;
      M_回原低速变更 : Bool;
      M_点动正速度变更 : Bool;
      M_点动负速度变更 : Bool;
      M_最高速度变更 : Bool;
      M_回原高速写入 : Bool;
      M_回原低速写入 : Bool;
      M_点动正速度写入 : Bool;
      M_点动负速度写入 : Bool;
      M_最高速度写入 : Bool;
      M_开始 : Bool;
      MW_Parameter : Int;
      MW_Index : Int;
      MD_Value : DInt;
      M_Pulse : Array[1..2] of Bool;
   END_VAR
   VAR_TEMP   // added for the SCL form of the ladder/FBD networks
      _w1 : Bool;
      _w2 : Bool;
      _w3 : Bool;
      _w4 : Bool;
      _w5 : Bool;
      _w6 : Bool;
   END_VAR
BEGIN

REGION Network 1: 回原高速
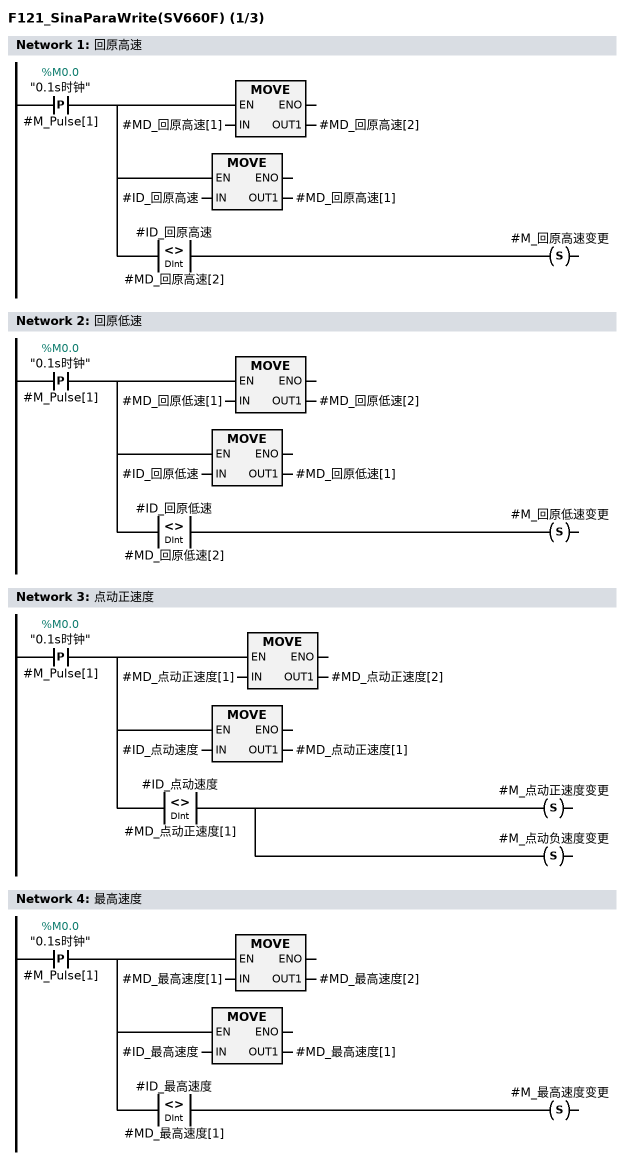
   RUNG wire#powerrail
      P_Contact(operand := "0.1s时钟", bit := #M_Pulse[1])
      wire#w1
      Move(in := #MD_回原高速[1], out1 => #MD_回原高速[2])
   END_RUNG
   RUNG wire#w1
      Move(in := #ID_回原高速, out1 => #MD_回原高速[1])
   END_RUNG
   RUNG wire#w1
      { S7_Templates := "SrcType := DInt" } NE_Contact(in1 := #ID_回原高速, in2 := #MD_回原高速[2])
      S_Coil( #M_回原高速变更 )
   END_RUNG
   // the same network as SCL:
   #_w1 := "0.1s时钟" AND NOT #M_Pulse[1];   // rising edge of "0.1s时钟"
   #M_Pulse[1] := "0.1s时钟";
   IF #_w1 THEN
       #MD_回原高速[2] := #MD_回原高速[1];
       #MD_回原高速[1] := #ID_回原高速;
   END_IF;
   IF #_w1 AND (#ID_回原高速 <> #MD_回原高速[2]) THEN #M_回原高速变更 := TRUE; END_IF;
END_REGION

REGION Network 2: 回原低速
   RUNG wire#powerrail
      P_Contact(operand := "0.1s时钟", bit := #M_Pulse[1])
      wire#w1
      Move(in := #MD_回原低速[1], out1 => #MD_回原低速[2])
   END_RUNG
   RUNG wire#w1
      Move(in := #ID_回原低速, out1 => #MD_回原低速[1])
   END_RUNG
   RUNG wire#w1
      { S7_Templates := "SrcType := DInt" } NE_Contact(in1 := #ID_回原低速, in2 := #MD_回原低速[2])
      S_Coil( #M_回原低速变更 )
   END_RUNG
   // the same network as SCL:
   #_w1 := "0.1s时钟" AND NOT #M_Pulse[1];   // rising edge of "0.1s时钟"
   #M_Pulse[1] := "0.1s时钟";
   IF #_w1 THEN
       #MD_回原低速[2] := #MD_回原低速[1];
       #MD_回原低速[1] := #ID_回原低速;
   END_IF;
   IF #_w1 AND (#ID_回原低速 <> #MD_回原低速[2]) THEN #M_回原低速变更 := TRUE; END_IF;
END_REGION

REGION Network 3: 点动正速度
   RUNG wire#powerrail
      P_Contact(operand := "0.1s时钟", bit := #M_Pulse[1])
      wire#w1
      Move(in := #MD_点动正速度[1], out1 => #MD_点动正速度[2])
   END_RUNG
   RUNG wire#w1
      Move(in := #ID_点动速度, out1 => #MD_点动正速度[1])
   END_RUNG
   RUNG wire#w1
      { S7_Templates := "SrcType := DInt" } NE_Contact(in1 := #ID_点动速度, in2 := #MD_点动正速度[1])
      wire#w2
      S_Coil( #M_点动正速度变更 )
   END_RUNG
   RUNG wire#w2
      S_Coil( #M_点动负速度变更 )
   END_RUNG
   // the same network as SCL:
   #_w1 := "0.1s时钟" AND NOT #M_Pulse[1];   // rising edge of "0.1s时钟"
   #M_Pulse[1] := "0.1s时钟";
   IF #_w1 THEN
       #MD_点动正速度[2] := #MD_点动正速度[1];
       #MD_点动正速度[1] := #ID_点动速度;
   END_IF;
   IF #_w1 AND (#ID_点动速度 <> #MD_点动正速度[1]) THEN
       #M_点动正速度变更 := TRUE;
       #M_点动负速度变更 := TRUE;
   END_IF;
END_REGION

REGION Network 4: 最高速度
   RUNG wire#powerrail
      P_Contact(operand := "0.1s时钟", bit := #M_Pulse[1])
      wire#w1
      Move(in := #MD_最高速度[1], out1 => #MD_最高速度[2])
   END_RUNG
   RUNG wire#w1
      Move(in := #ID_最高速度, out1 => #MD_最高速度[1])
   END_RUNG
   RUNG wire#w1
      { S7_Templates := "SrcType := DInt" } NE_Contact(in1 := #ID_最高速度, in2 := #MD_最高速度[1])
      S_Coil( #M_最高速度变更 )
   END_RUNG
   // the same network as SCL:
   #_w1 := "0.1s时钟" AND NOT #M_Pulse[1];   // rising edge of "0.1s时钟"
   #M_Pulse[1] := "0.1s时钟";
   IF #_w1 THEN
       #MD_最高速度[2] := #MD_最高速度[1];
       #MD_最高速度[1] := #ID_最高速度;
   END_IF;
   IF #_w1 AND (#ID_最高速度 <> #MD_最高速度[1]) THEN #M_最高速度变更 := TRUE; END_IF;
END_REGION

REGION Network 5
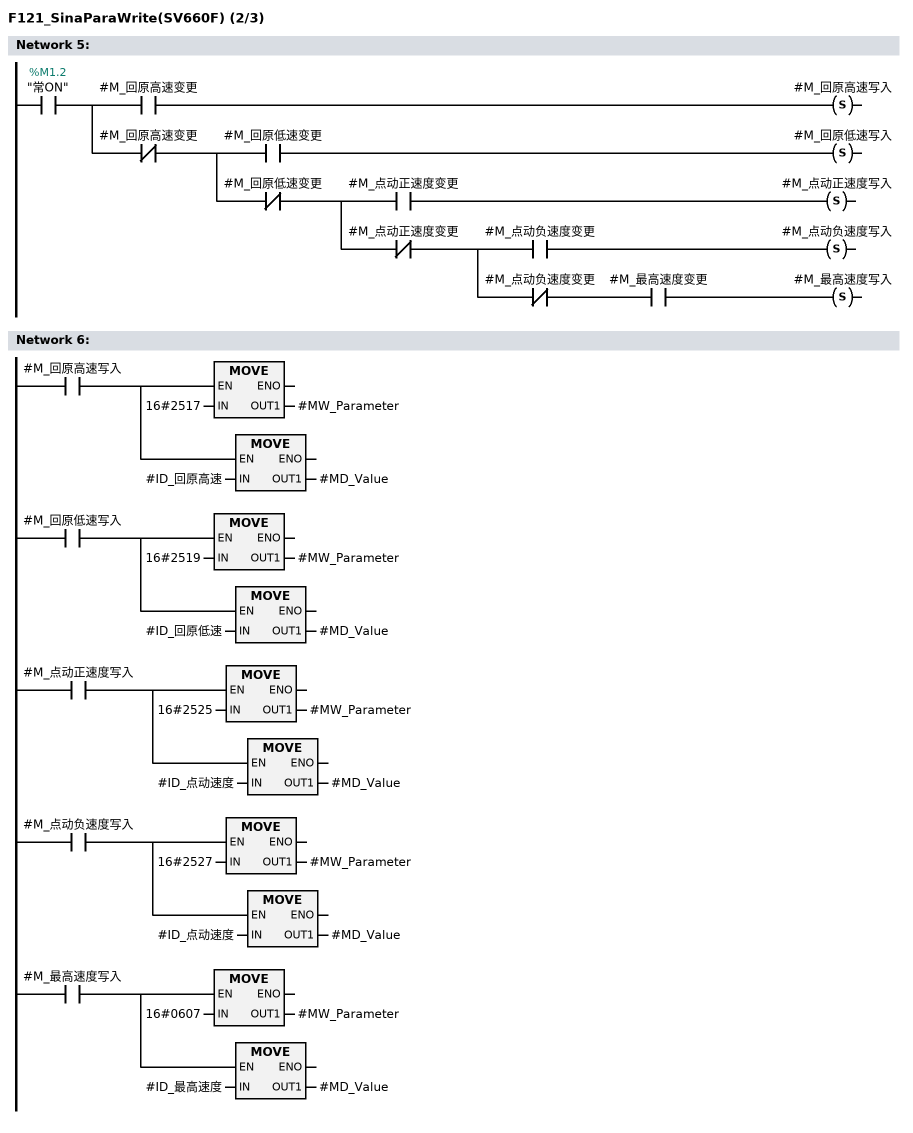
   RUNG wire#powerrail
      Contact( "常ON" )
      wire#w1
      Contact( #M_回原高速变更 )
      S_Coil( #M_回原高速写入 )
   END_RUNG
   RUNG wire#w1
      I_Contact( #M_回原高速变更 )
      wire#w2
      Contact( #M_回原低速变更 )
      S_Coil( #M_回原低速写入 )
   END_RUNG
   RUNG wire#w2
      I_Contact( #M_回原低速变更 )
      wire#w3
      Contact( #M_点动正速度变更 )
      S_Coil( #M_点动正速度写入 )
   END_RUNG
   RUNG wire#w3
      I_Contact( #M_点动正速度变更 )
      wire#w4
      Contact( #M_点动负速度变更 )
      S_Coil( #M_点动负速度写入 )
   END_RUNG
   RUNG wire#w4
      I_Contact( #M_点动负速度变更 )
      Contact( #M_最高速度变更 )
      S_Coil( #M_最高速度写入 )
   END_RUNG
   // the same network as SCL:
   IF "常ON" AND #M_回原高速变更 THEN #M_回原高速写入 := TRUE; END_IF;
   #_w1 := "常ON" AND NOT #M_回原高速变更;
   IF #_w1 AND #M_回原低速变更 THEN #M_回原低速写入 := TRUE; END_IF;
   #_w2 := #_w1 AND NOT #M_回原低速变更;
   IF #_w2 AND #M_点动正速度变更 THEN #M_点动正速度写入 := TRUE; END_IF;
   #_w3 := #_w2 AND NOT #M_点动正速度变更;
   IF #_w3 AND #M_点动负速度变更 THEN #M_点动负速度写入 := TRUE; END_IF;
   IF #_w3 AND NOT #M_点动负速度变更 AND #M_最高速度变更 THEN #M_最高速度写入 := TRUE; END_IF;
END_REGION

REGION Network 6
   RUNG wire#powerrail
      Contact( #M_回原高速写入 )
      wire#w1
      Move(in := 16#2517, out1 => #MW_Parameter)
   END_RUNG
   RUNG wire#w1
      Move(in := #ID_回原高速, out1 => #MD_Value)
   END_RUNG
   RUNG wire#powerrail
      Contact( #M_回原低速写入 )
      wire#w2
      Move(in := 16#2519, out1 => #MW_Parameter)
   END_RUNG
   RUNG wire#w2
      Move(in := #ID_回原低速, out1 => #MD_Value)
   END_RUNG
   RUNG wire#powerrail
      Contact( #M_点动正速度写入 )
      wire#w3
      Move(in := 16#2525, out1 => #MW_Parameter)
   END_RUNG
   RUNG wire#w3
      Move(in := #ID_点动速度, out1 => #MD_Value)
   END_RUNG
   RUNG wire#powerrail
      Contact( #M_点动负速度写入 )
      wire#w4
      Move(in := 16#2527, out1 => #MW_Parameter)
   END_RUNG
   RUNG wire#w4
      Move(in := #ID_点动速度, out1 => #MD_Value)
   END_RUNG
   RUNG wire#powerrail
      Contact( #M_最高速度写入 )
      wire#w5
      Move(in := 16#0607, out1 => #MW_Parameter)
   END_RUNG
   RUNG wire#w5
      Move(in := #ID_最高速度, out1 => #MD_Value)
   END_RUNG
   // the same network as SCL:
   IF #M_回原高速写入 THEN
       #MW_Parameter := 16#2517;
       #MD_Value := #ID_回原高速;
   END_IF;
   IF #M_回原低速写入 THEN
       #MW_Parameter := 16#2519;
       #MD_Value := #ID_回原低速;
   END_IF;
   IF #M_点动正速度写入 THEN
       #MW_Parameter := 16#2525;
       #MD_Value := #ID_点动速度;
   END_IF;
   IF #M_点动负速度写入 THEN
       #MW_Parameter := 16#2527;
       #MD_Value := #ID_点动速度;
   END_IF;
   IF #M_最高速度写入 THEN
       #MW_Parameter := 16#0607;
       #MD_Value := #ID_最高速度;
   END_IF;
END_REGION

REGION Network 7
